# B&R Automation Studio project dbserv_0640 (part 12)

#### brtcp.c
```c
#ifdef _DEFAULT_INCLUDES
	#include <AsDefault.h>
#endif
/*************************************************************************************************
	Treiber für TCP/IP-Kopplung zwischen zenOn und brserver

	Stand:		11.04.03
	Verfasser:	L.Waibel, MEGASYSTEMS GmbH
    LastEdit:

        21.12.04/RES:	#include von bsrun.h bzw. dbserv.h durch Compilerschalter geregelt
        11.12.04/RES:	Fehler bei ClientCommands() - case BRT_ITM_READ beseitigt
        08.12.03/Wai:	Fehler bei ITEM_WRITE ohne vorheriges LOGON behoben
		06.07.04/WAI:	Diagnose wegen Abstürzen mit divide-error
						(ClientDiag = protokollieren aller Client-Anmeldungen, ClientsMax=max.Anzahl Clients,
						Verwendung der max.Anzahl Clients aus dplist, statt MAX_CLIENTS
    	13.08.03/RES:	Diagnose-PVs reduziert; ClientDiagnose() eingefuegt ( nur fuer Burklimat2000 )
 		11.08.03/RES:	Alle "i" ersetzt durch "clientNr"
        15.07.03/RES:	Diagnosen eingebaut DIAG_*
                        Fehler bei ClientRecv() und ClientCommands() beseitigt
		08.09.06/WAI:	ClientConnect() Client möglichst wieder bei gleicher Instanz anmelden
						wegen Archivierung
		18.02.15/BIE:	Erweiterung für ATOM-CPUs

**************************************************************************************************/

#define _REPLACE_CONST		//18.02.2015 Erweiterung für ATOM-CPUs
#define ETH_SOCK_NG 1		//18.02.2015 Erweiterung für ATOM-CPUs

#include	<bur/plc.h>
#include	<bur/plctypes.h>
#include	<ethsock.h>
#include	<AsIecCon.h>
#include	<sys_lib.h>
#include	<standard.h>
#include 	<fileio.h>

#include	"platform.h"

#include	"brtcp.h"

#ifdef BURKLIMAT2000
			#include 	"bsrun.h"
			#include	"bksys.h"
#else
			#include	"dbserv.h"
#endif

/*************************************************************************************************/
/* Diagnose wegen Abstürzen */
#define	ANZAHL_CLIENTDIAG	10

typedef struct {
	UDINT		ClientAdrs;
	RTCtime_typ	LoginTime;
	UINT		LoginCount;
} CLIENTDIAG_typ;

_LOCAL	INT	ClientsMax,MaxCfgClients;
_LOCAL	CLIENTDIAG_typ	ClientDiag[ANZAHL_CLIENTDIAG];
_LOCAL	UINT	instancestate;
_LOCAL	RTCtime_typ	ActTime;

/*************************************************************************************************/
/*	globale Variablen                                                                            */
/*************************************************************************************************/

/*************************************************************************************************/
/*	lokale Variablen                                                                             */
/*************************************************************************************************/
_LOCAL	ACCESS_SERVER	*myidBrServer;

_LOCAL	UINT	idstat,brstate,portstat,timeoutstat,timeout;

_LOCAL	UINT	typestate,typecount;
_LOCAL	USINT 	step, initok;
_LOCAL	UINT	port;
_LOCAL	unsigned long	arg, socket_descr, bacllog, client_len;
_LOCAL	signed long	new_sock;
_LOCAL	int		opt_val, stat_ioctl, stat_setsockopt, stat_bind, stat_listen, clients;
_LOCAL	UINT	StateRTCTime,StateSWTime;
_LOCAL	INT		len_opt_val;

_LOCAL	ETH_sockaddr_typ name_str, client_str;
_LOCAL	INT	error;

_LOCAL	UINT	ID,AK,Anlage,Geraet,Typ,Punkt,Item;
_LOCAL	UDINT	Len,CmdLen,SendLen;

_LOCAL	CLI_HEAD_TYP *pBRT_head;
_LOCAL	CLI_LOGON_REQUEST *pBRT_logon;
_LOCAL	CLI_LOGON_RESPONSE *pBRT_logon_resp;
_LOCAL	CLI_LOGOFF_REQUEST *pBRT_logoff;
_LOCAL	CLI_LOGOFF_RESPONSE *pBRT_logoff_resp;
_LOCAL	CLI_READ_REQUEST *pBRT_read;
_LOCAL	CLI_READ_RESPONSE *pBRT_read_resp;
_LOCAL	CLI_WRITE_REQUEST *pBRT_write;
_LOCAL	CLI_WRITE_RESPONSE *pBRT_write_resp;
_LOCAL	CLI_ADRERROR_RESPONSE *pBRT_adrerror_resp;
_LOCAL	CLI_ERROR_RESPONSE *pBRT_error_resp;
_LOCAL	CLI_EVENT_RESPONSE *pBRT_event_resp;
_LOCAL	CLI_WATCHDOG_REQUEST *pBRT_watch;
_LOCAL	CLI_WATCHDOG_RESPONSE *pBRT_watch_resp;
_LOCAL	CLI_TIMESYNC_REQUEST *pBRT_time;
_LOCAL	CLI_TIMESYNC_RESPONSE *pBRT_time_resp;
_LOCAL	CLI_DATASTREAM *pBRT_datastream;

_LOCAL	client_typ	client[MAX_CLIENTS];
_LOCAL	USINT		TempBuffIn[RECVBUFLEN];
_LOCAL	USINT		TempBuffOut[SENDBUFLEN];
_LOCAL	USINT	DataByte;
_LOCAL	UINT	DataWord;
_LOCAL	UDINT	DataLong;
_LOCAL	RTCtime_typ DataTime;

_LOCAL	EVENT_PIPE_DATA	*pMSEventHeadData;

_LOCAL	unsigned char	DIAG_Init;
_LOCAL	unsigned long	DIAG_ClientAuftraege;
_LOCAL	unsigned long	DIAG_EventAuftraege;
_LOCAL	unsigned long	DIAG_LogonCount;

/***********************************************************************************************
	htons
	host to network short
***********************************************************************************************/
UINT htons(UINT in)
{
#ifndef INTEL
	return swapUINT(in);
#else
	return in;
#endif
}
/***********************************************************************************************
	htonl
	host to network long
***********************************************************************************************/
UDINT htonl(UDINT in)
{
#ifndef INTEL
	return swapUDINT(in);
#else
	return in;
#endif
}
/***********************************************************************************************
	ntohs
	network to host short
***********************************************************************************************/
UINT ntohs(UINT in)
{
#ifndef INTEL
	return swapUINT(in);
#else
	return in;
#endif
}

/***********************************************************************************************
	ntohl
	network to host long
***********************************************************************************************/
UDINT ntohl(UDINT in)
{
#ifndef INTEL
	return swapUDINT(in);
#else
	return in;
#endif
}
/***********************************************************************************************
	GetData
	kopiert plattformabhägig die Daten und stellt die korrekte Byte-Order her
	Rückgabe:	Zeiger auf die korrekten Daten
***********************************************************************************************/
void GetData( USINT *pDataSrc, USINT **pDataDest, UDINT Len)
{
	switch(Len)	{
		default:
		case 1:
			DataByte = *(USINT*)pDataSrc;
			*pDataDest = &DataByte;
			break;
		case 2:
			DataWord = ntohs(*(UINT*)pDataSrc);
			*pDataDest = (USINT*)&DataWord;
			break;
		case 4:
			DataLong = ntohl(*(UDINT*)pDataSrc);
			*pDataDest = (USINT*)&DataLong;
			break;
		case sizeof(RTCtime_typ):
			memcpy((USINT*)&DataTime,pDataSrc,Len);
			DataTime.year = ntohs(DataTime.year);
			*pDataDest = (USINT*)&DataTime;
			break;
	}
}

/***********************************************************************************************
	TcpError
	kodiert die Meldeserver-Fehlernummern auf TCP-Fehlernummern um
***********************************************************************************************/
UINT TcpError(UINT inerror)
{
	UINT	outerror;

	switch (inerror)	{
		case cEC_INVALID_UNIT:
			outerror = BRT_ERR_UNKNOWN_UNIT;
			break;
		case cEC_INVALID_DEVICE:
			outerror = BRT_ERR_UNKNOWN_DEVICE;
			break;
		case cEC_INVALID_TYPE:
			outerror = BRT_ERR_UNKNOWN_TYPE;
			break;
		case cEC_INVALID_POINT:
			outerror = BRT_ERR_UNKNOWN_POINT;
			break;
		case cEC_INVALID_ITEM:
			outerror = BRT_ERR_WRONG_ITEM;
			break;
		case cEC_INVALID_LENGTH:
			outerror = BRT_ERR_WRONG_LEN;
			break;
		case cEC_ITEM_ALREADY_LINKED:
			outerror = BRT_ERR_IS_LOGGED;
			break;
		case cEC_ITEM_ALREADY_UNLINKED:
			outerror = BRT_ERR_ITEM_NO_LOGON;
			break;
		case cEC_ITEM_NOT_WRITEABLE:
			outerror = BRT_ERR_ITEM_NOT_WRITEABLE;
			break;
		case cEC_WRITE_PIPE_FULL:
			outerror = BRT_ERR_WRITE_PIPE_FULL;
			break;
		case cEC_ITEM_NO_TIMESTAMP:
			outerror = BRT_ERR_ITEM_NO_TS;
			break;
		case cEC_INVALID_VALUE:
			outerror = BRT_ERR_ITEM_NO_DATA;
			break;
		default:
			outerror = inerror;
			break;
	}
	return outerror;
}
/***********************************************************************************************
	GetAdrs
	liest die aktuelle Adresse aus dem Telegramm in Einzelvariablen
***********************************************************************************************/
void GetAdrs(CLI_ADR_TYP *pAdrs)
{
	Anlage = ntohs(pAdrs->anlage);
	Geraet = ntohs(pAdrs->geraet);
	Typ = ntohs(pAdrs->typ);
	Punkt = ntohs(pAdrs->punkt);
	Item = ntohs(pAdrs->item);
}
/***********************************************************************************************
	PutAdrs
	schreibt die aktuelle Adresse in das Telegramm aus Einzelvariablen
***********************************************************************************************/
void PutAdrs(CLI_ADR_TYP *pAdrs)
{
	pAdrs->anlage = htons(Anlage);
	pAdrs->geraet = htons(Geraet);
	pAdrs->typ = htons(Typ);
	pAdrs->punkt = htons(Punkt);
	pAdrs->item = htons(Item);
}
/***********************************************************************************************
	NextCmd
	schaltet Empfangspuffer auf nächsten Befehl und setzt ggf. Puffer zurück
***********************************************************************************************/
void NextCmd(INT clientNr, UDINT len)
{
	client[clientNr].recv_out += len;
	if(client[clientNr].recv_out == client[clientNr].recv_in)	{
		client[clientNr].recv_out = client[clientNr].recv_in = 0;		/* reset buffer */
	}
}
/***********************************************************************************************
	SpaceSendBuf
	prüft, ob die angeforderte Datenlänge noch in den Sendepuffer passt
***********************************************************************************************/
int SpaceSendBuf(INT clientNr, UDINT len)
{
	return( (sizeof(client[clientNr].send_buf) - client[clientNr].send_in) > len ? 1:0);
}

/***********************************************************************************************
	ClientConnect
	akzeptiert neue Client-Verbindungen
***********************************************************************************************/
void ClientConnect()
{
	INT	clientNr;
	BOOL new_client;
	BOOL old_entry;

	new_client = FALSE;
	client_len = sizeof(client_str);
	new_sock = accept(socket_descr, (unsigned long)&client_str, (unsigned long)&client_len);
	if (new_sock != ERR_SOCKET)	{
		/* new connection */
		for(clientNr=0;clientNr<MaxCfgClients;clientNr++)	{		/* 06.07.04: statt MAX_CLIENTS */
			/* 08.09.06: gleichen Client über IP-Adrs möglichst an gleicher Instanz anmelden wegen Archivierung */
			if(client[clientNr].socket==ERR_SOCKET && client[clientNr].client_str.sin_addr == client_str.sin_addr)	{
				/* new client */
				client[clientNr].socket = new_sock;
				client[clientNr].recv_in = 0;
				client[clientNr].recv_out = 0;
				client[clientNr].send_in = 0;
				client[clientNr].send_out = 0;
				client[clientNr].status = CLI_CONNECTED;
				client[clientNr].TON_watchdog.IN = FALSE;
				client[clientNr].stateEvRead = cEC_NO_DATA_IN_EVENTBUFFER;
				clients++;
				/* 06.07.04: save ClientsMax */
				if(clients > ClientsMax)	ClientsMax = clients;

				new_client = TRUE;
				memcpy(&client[clientNr].client_str,&client_str,sizeof(client_str));
				break;
			}
		}
		if(!new_client)	{
			/* 08.09.06: falls Client noch nie angemeldet war: nächsten freien Client nehmen */
			for(clientNr=0;clientNr<MaxCfgClients;clientNr++)	{		/* 06.07.04: statt MAX_CLIENTS */
				if(client[clientNr].socket==ERR_SOCKET)	{
					/* new client */
					client[clientNr].socket = new_sock;
					client[clientNr].recv_in = 0;
					client[clientNr].recv_out = 0;
					client[clientNr].send_in = 0;
					client[clientNr].send_out = 0;
					client[clientNr].status = CLI_CONNECTED;
					client[clientNr].TON_watchdog.IN = FALSE;
					client[clientNr].stateEvRead = cEC_NO_DATA_IN_EVENTBUFFER;
					clients++;
					/* ArchiveFiles löschen bei neuem Client */

					/* 06.07.04: save ClientsMax */
					if(clients > ClientsMax)	ClientsMax = clients;

					new_client = TRUE;
					memcpy(&client[clientNr].client_str,&client_str,sizeof(client_str));
					break;
				}
			}
		}
		/*---------------------------------------------------------------------------*/
		/* 06.07.04: diagnostics: log every connecting client */
		old_entry = 0;
		for(clientNr=0;clientNr< ANZAHL_CLIENTDIAG;clientNr++)	{
			if(ClientDiag[clientNr].ClientAdrs == client_str.sin_addr)	{
				RTC_gettime(&ActTime);
				memcpy(&ClientDiag[clientNr].LoginTime,&ActTime,sizeof(ActTime));
				ClientDiag[clientNr].LoginCount++;
				old_entry = TRUE;
				break;
			}
		}
		if(!old_entry)	{
			/* look for new entry in list */
			for(clientNr=0;clientNr< ANZAHL_CLIENTDIAG;clientNr++)	{
				if(ClientDiag[clientNr].ClientAdrs == 0 || clientNr == ANZAHL_CLIENTDIAG-1)	{	/* auf jeden in letztem Platz eintragen */
					RTC_gettime(&ActTime);
					ClientDiag[clientNr].ClientAdrs = client_str.sin_addr;
					memcpy(&ClientDiag[clientNr].LoginTime,&ActTime,sizeof(ActTime));
					ClientDiag[clientNr].LoginCount++;
					break;
				}
			}
		}
		/* 06.07.04: end diagnostics: log every connecting client */
		/*---------------------------------------------------------------------------*/

		if(!new_client)	{
			close(new_sock);		/* immediately terminate new connection */
		}
	}
}
/***********************************************************************************************
	ClientClose
	beendet Verbindung zu einem Client
***********************************************************************************************/
void ClientClose(INT clientNr, INT reason)
{
	close(client[clientNr].socket);
	client[clientNr].socket = ERR_SOCKET;
	client[clientNr].status = reason;
	client[clientNr].TON_watchdog.IN = FALSE;
/*	UnlinkEventInstance(myidBrServer,clientNr);*/
	UnlinkEventInstanceWithoutFileBuffer(myidBrServer,clientNr);		/* WAI 09.04.06 */
	if(clients)	clients--;
}
/***********************************************************************************************
	ClientWatch
	prüft auf Verbindungstimeout zu einem Client
***********************************************************************************************/
void ClientWatch(INT clientNr)
{
	TON(&client[clientNr].TON_watchdog);
	client[clientNr].TON_watchdog.IN = TRUE;
	if(client[clientNr].TON_watchdog.Q == TRUE)	{
		/* Timeout !	close connection */
		ClientClose(clientNr,CLI_WATCHDOG);
	}
}

/***********************************************************************************************
	ClientRecv
	empfängt Daten von den aktiven Clients
***********************************************************************************************/
UDINT ClientRecv(INT clientNr)
{
	DINT	bytes = 0;		/* 15.07.03/RES: bytes = 0 */
	UDINT	recv_len;

	/* read data from client */
	recv_len = sizeof(client[clientNr].recv_buf) - client[clientNr].recv_in;
	if( recv_len > 0 ) {		/* 15.07.03/RES */
		bytes = recv(client[clientNr].socket,(UDINT)&client[clientNr].recv_buf[client[clientNr].recv_in],recv_len,0);
		if(bytes==0)	{
			/* connection closed */
			ClientClose(clientNr,CLI_DISCONNECTED);
		}
		else if(bytes == ERR_SOCKET){
			/* error */
			error = EthGetError();
			if(error != ERR_ETH_WOULDBLOCK )	{
				/* all errors except: waiting for data */
				ClientClose(clientNr,CLI_ERROR);
			}
		}
		else {
			/* data received */
			client[clientNr].recv_cnt++;
			client[clientNr].TON_watchdog.IN = FALSE;
			client[clientNr].recv_in +=bytes;
		}
	}
	return bytes;
}
/***********************************************************************************************
	ClientCommands
	wertet die Kommandos eines Clients aus
***********************************************************************************************/
void ClientCommands(INT clientNr)
{
	BOOL	wait_data = FALSE;
	UDINT	shiftlen,TempLen;
	UINT	mserror = 0;
	USINT	*pData,*pTime,*pDest;
	UDINT	lenData,lenTime;

	if(client[clientNr].recv_in  < (client[clientNr].recv_out+sizeof(CLI_HEAD_TYP))) {
		wait_data = TRUE;		/* no data */
	}
	else {
		do	{

			memcpy(TempBuffIn,&client[clientNr].recv_buf[client[clientNr].recv_out],client[clientNr].recv_in - client[clientNr].recv_out);
			pBRT_head = (CLI_HEAD_TYP *)TempBuffIn;
			ID  = ntohs(pBRT_head->ID);
			AK	= ntohs(pBRT_head->AK);

			DIAG_ClientAuftraege++;

			switch(AK)	{
				/*...........................................................................................*/
				/* Item mit/ohne Zeitstempel anmelden */
				case BRT_ITM_LOGON:
				case BRT_ITM_LOGON_TS:
					if(client[clientNr].recv_in  >= (client[clientNr].recv_out+sizeof(CLI_LOGON_REQUEST)-2))	{
						pBRT_logon = (CLI_LOGON_REQUEST *)pBRT_head;
						Len = (UDINT)ntohs(pBRT_logon->LenHigh)<<16 | ntohs(pBRT_logon->LenLow) ;
						CmdLen = sizeof(CLI_LOGON_REQUEST)+ Len - 2;
						if(client[clientNr].recv_in  >= client[clientNr].recv_out + CmdLen)	{
							GetAdrs(&pBRT_logon->Adr);		/* Adresse aus Telegramm lesen */

							if(AK == BRT_ITM_LOGON)
								SendLen = CmdLen;						/* LOGON_RESPONSE max. gleich lang wie REQUEST ! */
							else
								SendLen = CmdLen +sizeof(RTCtime_typ);	/* LOGON_RESPONSE max. gleich lang wie REQUEST ! */

							if(SpaceSendBuf(clientNr, SendLen))	{	/* Platz in Sendepuffer vorhanden ?*/

								DIAG_LogonCount++;

								/* Hysterese kopieren */
								GetData((USINT*)&pBRT_logon->Data,(USINT**)&pData,Len);	/* Daten ggf. swappen */
								if((mserror = SetHystItem (myidBrServer,clientNr,Anlage,Geraet,Typ,Punkt,Item,pData,Len))==0)	{
									/* Datenpunkt anmelden */
									mserror=LinkEventItem(myidBrServer,clientNr,Anlage,Geraet,Typ,Punkt,Item,(AK == BRT_ITM_LOGON ? 0:1));
									if(mserror == 0 || mserror == cEC_ITEM_ALREADY_LINKED_FILE_BUFFER)	{	/* wegen Langzeitarchivierung */
										/* AktWert besorgen */
										mserror = GetValueItem (myidBrServer,clientNr, Anlage, Geraet, Typ, Punkt, Item, &pData, &lenData, &pTime, &lenTime);
									}
									if(mserror == 0)	{
										if( Len != lenData || (AK==BRT_ITM_LOGON_TS && lenTime==0))	{
											/* falsche Länge oder kein Zeitstempel vorhanden */
											if(Len != lenData)	mserror = BRT_ERR_WRONG_LEN;
											else				mserror = BRT_ERR_ITEM_NO_TS;

											pBRT_adrerror_resp = (CLI_ADRERROR_RESPONSE *)TempBuffOut;
											pBRT_adrerror_resp->head.ID = htons(ID);
											pBRT_adrerror_resp->head.AK = htons(BRT_ITM_LOGON_ERR);
											PutAdrs(&pBRT_adrerror_resp->Adr);
											pBRT_adrerror_resp->Error = htons(TcpError(mserror));
											SendLen = sizeof(CLI_ADRERROR_RESPONSE);
										}
										else {
											/* Sendedaten bereitstellen */
											pBRT_logon_resp = (CLI_LOGON_RESPONSE *)&TempBuffOut;
											pBRT_logon_resp->head.ID = htons(ID);
											PutAdrs(&pBRT_logon_resp->Adr);

											if(AK == BRT_ITM_LOGON)	{
												pBRT_logon_resp->head.AK = htons(BRT_ITM_LOGON_OK);
											}
											else	{
												pBRT_logon_resp->head.AK = htons(BRT_ITM_LOGON_TS_OK);
											}
											TempLen = htonl(lenData);
											memcpy(&pBRT_logon_resp->LenLow,&TempLen,sizeof(TempLen));
											/* Daten kopieren */
											GetData(pData,(USINT**)&pDest,lenData);
											memcpy(&pBRT_logon_resp->Data,pDest,lenData);
											/* ggf. Zeitstempel kopieren */
											if(AK == BRT_ITM_LOGON_TS)	{
												GetData(pTime,(USINT**)&pDest,lenTime);
												memcpy((USINT*)&pBRT_logon_resp->Data+lenData,pDest,lenTime);
											}
										}
									}
									else {	/* Fehler beim Lesen des Datenpunkts */
										/* Sendedaten bereitstellen */
										pBRT_adrerror_resp = (CLI_ADRERROR_RESPONSE *)TempBuffOut;
										pBRT_adrerror_resp->head.ID = htons(ID);
										pBRT_adrerror_resp->head.AK = htons(BRT_ITM_LOGON_ERR);
										PutAdrs(&pBRT_adrerror_resp->Adr);
										pBRT_adrerror_resp->Error = htons(TcpError(mserror));
										SendLen = sizeof(CLI_ADRERROR_RESPONSE);
									}
								}
								else {	/* logon-error */
									/* Sendedaten bereitstellen */
									pBRT_adrerror_resp = (CLI_ADRERROR_RESPONSE *)TempBuffOut;
									pBRT_adrerror_resp->head.ID = htons(ID);
									pBRT_adrerror_resp->head.AK = htons(BRT_ITM_LOGON_ERR);
									PutAdrs(&pBRT_adrerror_resp->Adr);
									pBRT_adrerror_resp->Error = htons(TcpError(mserror));

									SendLen = sizeof(CLI_ADRERROR_RESPONSE);
								}
								memcpy(&client[clientNr].send_buf[client[clientNr].send_in],TempBuffOut,SendLen);
								client[clientNr].send_in += SendLen;
								/* goto next command */
								NextCmd(clientNr, CmdLen);
							}
							else	wait_data = TRUE;	/* wait for sendbuffer free */
						}
						else wait_data = TRUE;	/* incomplete data */
					}
					else wait_data = TRUE;	/* incomplete data */
					break;
				/*...........................................................................................*/
				/* Item abmelden */
				case BRT_ITM_LOGOFF:
					CmdLen = sizeof(CLI_LOGOFF_REQUEST);
					if(client[clientNr].recv_in  >= client[clientNr].recv_out + CmdLen)	{
						pBRT_logoff = (CLI_LOGOFF_REQUEST *)pBRT_head;
						GetAdrs(&pBRT_logoff->Adr);		/* Adresse aus Telegramm lesen */

						SendLen = sizeof(CLI_ADRERROR_RESPONSE);	/* LOGOFF_RESPONSE max. gleich lang wie ADRERROR_RESPONSE ! */

						if(SpaceSendBuf(clientNr, SendLen))	{	/* Platz in Sendepuffer vorhanden ?*/
							if((error=UnlinkEventItem(myidBrServer,clientNr,Anlage,Geraet,Typ,Punkt,Item))==0)	{
								/* Sendedaten bereitstellen */
								pBRT_logoff_resp = (CLI_LOGOFF_RESPONSE *)TempBuffOut;
								pBRT_logoff_resp->head.ID = htons(ID);
								pBRT_logoff_resp->head.AK = htons(BRT_ITM_LOGOFF_OK);
								PutAdrs(&pBRT_logoff_resp->Adr);
								SendLen = CmdLen;
							}
							else {	/* logoff-error */
								/* Sendedaten bereitstellen */
								pBRT_adrerror_resp = (CLI_ADRERROR_RESPONSE *)TempBuffOut;
								pBRT_adrerror_resp->head.ID = htons(ID);
								pBRT_adrerror_resp->head.AK = htons(BRT_ITM_LOGOFF_ERR);
								PutAdrs(&pBRT_adrerror_resp->Adr);
								pBRT_adrerror_resp->Error = htons(TcpError(error));
								SendLen = sizeof(CLI_ADRERROR_RESPONSE);
							}
							memcpy(&client[clientNr].send_buf[client[clientNr].send_in],TempBuffOut,SendLen);
							client[clientNr].send_in += SendLen;
							/* goto next command */
							NextCmd(clientNr, CmdLen);
						}
						else	wait_data = TRUE;	/* wait for sendbuffer free */
					}
					else wait_data = TRUE;	/* incomplete data */
					break;
				/*...........................................................................................*/
				/* Item mit/ohne Zeitstempel lesen */
				case BRT_ITM_READ:
				case BRT_ITM_READ_TS:
					CmdLen = sizeof(CLI_READ_REQUEST);
					if(client[clientNr].recv_in  >= client[clientNr].recv_out + CmdLen)	{
						pBRT_read = (CLI_READ_REQUEST *)pBRT_head;
						GetAdrs(&pBRT_read->Adr);		/* Adresse aus Telegramm lesen */

						/* AktWert besorgen */
						mserror = GetValueItem (myidBrServer,clientNr, Anlage, Geraet, Typ, Punkt, Item, &pData, &lenData, &pTime, &lenTime);
						if(mserror == 0)	{
							if(AK==BRT_ITM_READ)
								SendLen = sizeof(CLI_READ_RESPONSE)+lenData-2;
							else
								SendLen = sizeof(CLI_READ_RESPONSE)+lenData-2+sizeof(RTCtime_typ);

							if(SpaceSendBuf(clientNr, SendLen))	{	/* Platz in Sendepuffer vorhanden ?*/
								if(AK==BRT_ITM_READ_TS && lenTime==0)	{
								/* kein Zeitstempel vorhanden */
									mserror = BRT_ERR_ITEM_NO_TS;

									pBRT_adrerror_resp = (CLI_ADRERROR_RESPONSE *)TempBuffOut;
									pBRT_adrerror_resp->head.ID = htons(ID);
									pBRT_adrerror_resp->head.AK = htons(BRT_ITM_READ_ERR);
									PutAdrs(&pBRT_adrerror_resp->Adr);
									pBRT_adrerror_resp->Error = htons(TcpError(mserror));
									SendLen = sizeof(CLI_ADRERROR_RESPONSE);
								}
								else {
									/* Sendedaten bereitstellen */
									pBRT_read_resp = (CLI_READ_RESPONSE *)&TempBuffOut;
									pBRT_read_resp->head.ID = htons(ID);
									PutAdrs(&pBRT_read_resp->Adr);

									if(AK == BRT_ITM_READ)	{
										pBRT_read_resp->head.AK = htons(BRT_ITM_READ_OK);
									}
									else	{
										pBRT_read_resp->head.AK = htons(BRT_ITM_READ_TS_OK);
										Len += sizeof(RTCtime_typ);
									}
									TempLen = htonl(lenData);	/* wegen alignment UDINT ! */
									memcpy(&pBRT_read_resp->LenLow,&TempLen,sizeof(TempLen));
									/* Daten kopieren */
									GetData(pData,(USINT**)&pDest,lenData);
									memcpy(&pBRT_read_resp->Data,pDest,lenData);
									/* ggf. Zeitstempel kopieren */
									if(AK == BRT_ITM_READ_TS) {						/* 11.12.04/RES: hier fehlende Klammern eingefuegt !! */
										GetData(pTime,(USINT**)&pDest,lenTime);
										memcpy((USINT*)&pBRT_read_resp->Data+lenData,pDest,lenTime);
									}
								}
								memcpy(&client[clientNr].send_buf[client[clientNr].send_in],TempBuffOut,SendLen);
								client[clientNr].send_in += SendLen;
								/* goto next command */
								NextCmd(clientNr, CmdLen);
							}
							else wait_data = TRUE;	/* wait for sendbuffer free */
						}
						else	{	/* Fehler beim Lesen des Datenpunkts */
							SendLen = sizeof(CLI_ADRERROR_RESPONSE);
							if(SpaceSendBuf(clientNr, SendLen))	{	/* Platz in Sendepuffer vorhanden ?*/
								pBRT_adrerror_resp = (CLI_ADRERROR_RESPONSE *)TempBuffOut;
								pBRT_adrerror_resp->head.ID = htons(ID);
								pBRT_adrerror_resp->head.AK = htons(BRT_ITM_LOGON_ERR);
								PutAdrs(&pBRT_adrerror_resp->Adr);
								pBRT_adrerror_resp->Error = htons(TcpError(mserror));

								memcpy(&client[clientNr].send_buf[client[clientNr].send_in],TempBuffOut,SendLen);
								client[clientNr].send_in += SendLen;
								/* goto next command */
								NextCmd(clientNr, CmdLen);
							}
							else wait_data = TRUE;	/* wait for sendbuffer free */
						}
					}
					else wait_data = TRUE;	/* incomplete data */
					break;
				/*...........................................................................................*/
				/* Item schreiben */
				case BRT_ITM_WRITE:
					if(client[clientNr].recv_in  >= (client[clientNr].recv_out+sizeof(CLI_WRITE_REQUEST)-2))	{
						pBRT_write = (CLI_WRITE_REQUEST *)pBRT_head;
						Len = (UDINT)ntohs(pBRT_write->LenHigh)<<16 | ntohs(pBRT_write->LenLow) ;
						CmdLen = sizeof(CLI_WRITE_REQUEST)+ Len - 2;
						if(client[clientNr].recv_in  >= client[clientNr].recv_out + CmdLen)	{
							GetAdrs(&pBRT_write->Adr);		/* Adresse aus Telegramm lesen */

							SendLen = sizeof(CLI_ADRERROR_RESPONSE);	/* WRITE_RESPONSE max. gleich lang wie ADRERROR_RESPONSE ! */

							if(SpaceSendBuf(clientNr, SendLen))	{	/* Platz in Sendepuffer vorhanden ?*/
								GetData((USINT*)&pBRT_write->Data,(USINT**)&pData,Len);	/* Daten ggf. swappen */
								mserror = SetWriteItem(myidBrServer,Anlage,Geraet,Typ,Punkt,Item,pData,Len);

								if(mserror==0)	{
									/* Sendedaten bereitstellen */
									pBRT_write_resp = (CLI_WRITE_RESPONSE *)TempBuffOut;
									pBRT_write_resp->head.ID = htons(ID);
									PutAdrs(&pBRT_write_resp->Adr);
									pBRT_write_resp->head.AK = htons(BRT_ITM_WRITE_OK);
									SendLen = sizeof(CLI_WRITE_RESPONSE);
								}
								else {	/* write-error */
									/* Sendedaten bereitstellen */
									pBRT_adrerror_resp = (CLI_ADRERROR_RESPONSE *)TempBuffOut;
									pBRT_adrerror_resp->head.ID = htons(ID);
									pBRT_adrerror_resp->head.AK = htons(BRT_ITM_WRITE_ERR);
									PutAdrs(&pBRT_adrerror_resp->Adr);
									pBRT_adrerror_resp->Error = htons(TcpError(mserror));
									SendLen = sizeof(CLI_ADRERROR_RESPONSE);
								}
								memcpy(&client[clientNr].send_buf[client[clientNr].send_in],TempBuffOut,SendLen);
								client[clientNr].send_in += SendLen;
								/* goto next command */
								NextCmd(clientNr, CmdLen);
							}
							else	wait_data = TRUE;	/* wait for sendbuffer free */
						}
						else wait_data = TRUE;	/* incomplete data */
					}
					else wait_data = TRUE;	/* incomplete data */
					break;
				/*...........................................................................................*/
				/* Datenstrom lesen */
				case BRT_DATASTREAM_READ:
					CmdLen = sizeof(CLI_READ_REQUEST);
					if(client[clientNr].recv_in  >= client[clientNr].recv_out + CmdLen)	{
						pBRT_read = (CLI_READ_REQUEST *)pBRT_head;
						GetAdrs(&pBRT_read->Adr);		/* Adresse aus Telegramm lesen */

						/* Sonderbehandlung fehlt noch . eigener Buffer, eigenes Flag .. */
						/* AktWert besorgen */
						/*mserror = get_station_type_point (idMessageServer, Geraet, Typ, Punkt, &pData, &lenData, 0, 0, &pTime, &lenTime, 0, 0);*/
						if(mserror == 0)	{
							SendLen = sizeof(CLI_READ_RESPONSE)+lenData-2;

							if(SpaceSendBuf(clientNr, SendLen))	{	/* Platz in Sendepuffer vorhanden ?*/
								/* Sendedaten bereitstellen */
								pBRT_read_resp = (CLI_READ_RESPONSE *)&TempBuffOut;
								pBRT_read_resp->head.ID = htons(ID);
								PutAdrs(&pBRT_read_resp->Adr);

								pBRT_read_resp->head.AK = htons(BRT_DATASTREAM_READ_OK);

								TempLen = htonl(lenData);	/* wegen alignment UDINT ! */
								memcpy(&pBRT_read_resp->LenLow,&TempLen,sizeof(TempLen));
								/* Daten kopieren */
								memcpy(&pBRT_read_resp->Data,pData,lenData);

								memcpy(&client[clientNr].send_buf[client[clientNr].send_in],TempBuffOut,SendLen);
								client[clientNr].send_in += SendLen;
								/* goto next command */
								NextCmd(clientNr, CmdLen);
							}
							else wait_data = TRUE;	/* wait for sendbuffer free */
						}
						else	{	/* Fehler beim Lesen des Datenpunkts */
							SendLen = sizeof(CLI_ADRERROR_RESPONSE);
							if(SpaceSendBuf(clientNr, SendLen))	{	/* Platz in Sendepuffer vorhanden ?*/
								pBRT_adrerror_resp = (CLI_ADRERROR_RESPONSE *)TempBuffOut;
								pBRT_adrerror_resp->head.ID = htons(ID);
								pBRT_adrerror_resp->head.AK = htons(BRT_DATASTREAM_READ_ERR);
								PutAdrs(&pBRT_adrerror_resp->Adr);
								pBRT_adrerror_resp->Error = htons(TcpError(mserror));
							}
							else wait_data = TRUE;	/* wait for sendbuffer free */
						}
					}
					else wait_data = TRUE;	/* incomplete data */
					break;
				/*...........................................................................................*/
				/* Watchdog */
				case BRT_CLI_WATCHDOG:
					CmdLen = sizeof(CLI_WATCHDOG_REQUEST);
					if(client[clientNr].recv_in  >= client[clientNr].recv_out + CmdLen)	{
						pBRT_watch = (CLI_WATCHDOG_REQUEST *)pBRT_head;
						SendLen = sizeof(CLI_WATCHDOG_RESPONSE);

						if(SpaceSendBuf(clientNr, SendLen))	{	/* Platz in Sendepuffer vorhanden ?*/
							/* Sendedaten bereitstellen */
							pBRT_watch_resp = (CLI_WATCHDOG_RESPONSE *)TempBuffOut;
							pBRT_watch_resp->head.ID = htons(ID);
							pBRT_watch_resp->head.AK = htons(BRT_CLI_WATCHDOG_OK);
							memcpy(&client[clientNr].send_buf[client[clientNr].send_in],TempBuffOut,SendLen);
							client[clientNr].send_in += SendLen;
							/* goto next command */
							NextCmd(clientNr, CmdLen);
						}
						else	wait_data = TRUE;	/* wait for sendbuffer free */
					}
					else wait_data = TRUE;	/* incomplete data */
					break;
				/*...........................................................................................*/
				/* Zeitsynchronisation */
				case BRT_TIMESYNC:
					CmdLen = sizeof(CLI_TIMESYNC_REQUEST);
					if(client[clientNr].recv_in  >= client[clientNr].recv_out + CmdLen)	{
						pBRT_time = (CLI_TIMESYNC_REQUEST *)pBRT_head;
						SendLen = sizeof(CLI_ERROR_RESPONSE);		/* max.Antwortlänge */

						if(SpaceSendBuf(clientNr, SendLen))	{	/* Platz in Sendepuffer vorhanden ?*/
							/* Echtzeituhr stellen */
							pBRT_time->Time.year = ntohs(pBRT_time->Time.year );
							pBRT_time->Time.reserve = 0;
/*							pBRT_time->Time.millisec = 0;
							pBRT_time->Time.microsec = 0;*/
							StateRTCTime = RTC_settime(&pBRT_time->Time);
	#ifndef INTEL
							StateSWTime = SW_settime(&pBRT_time->Time);
	#else
							StateSWTime = 0;
	#endif

							if(StateRTCTime==0 && StateSWTime==0)	{
								/* Sendedaten bereitstellen */
								pBRT_time_resp = (CLI_TIMESYNC_RESPONSE *)TempBuffOut;
								pBRT_time_resp->head.ID = htons(ID);
								pBRT_time_resp->head.AK = htons(BRT_TIMESYNC_OK);
								SendLen = sizeof(CLI_TIMESYNC_RESPONSE );
							}
							else {	/* Fehler bei Uhrzeit stellen */
								pBRT_error_resp = (CLI_ERROR_RESPONSE *)TempBuffOut;
								pBRT_error_resp->head.ID = htons(ID);
								pBRT_error_resp->head.AK = htons(BRT_TIMESYNC_ERR);
								if(StateRTCTime)	pBRT_error_resp->Error = htons(BRT_ERR_RTC_SET);
								else				pBRT_error_resp->Error = htons(BRT_ERR_SWC_SET);
							}
							memcpy(&client[clientNr].send_buf[client[clientNr].send_in],TempBuffOut,SendLen);
							client[clientNr].send_in += SendLen;
							/* goto next command */
							NextCmd(clientNr, CmdLen);
						}
						else	wait_data = TRUE;	/* wait for sendbuffer free */
					}
					else wait_data = TRUE;	/* incomplete data */
					break;
				/*...........................................................................................*/
				/* unbekannte Auftragskennung */
				default:
					SendLen = sizeof(CLI_ERROR_RESPONSE);

					if(SpaceSendBuf(clientNr, SendLen))	{	/* Platz in Sendepuffer vorhanden ?*/
						/* Sendedaten bereitstellen */
						pBRT_error_resp = (CLI_ERROR_RESPONSE *)TempBuffOut;
						pBRT_error_resp->head.ID = htons(ID);
						pBRT_error_resp->head.AK = htons(BRT_CLI_ERROR);
						error = BRT_ERR_INVALIDAK;
						pBRT_error_resp->Error = htons(error);
						SendLen = sizeof(CLI_ERROR_RESPONSE);
						memcpy(&client[clientNr].send_buf[client[clientNr].send_in],TempBuffOut,SendLen);
						client[clientNr].send_in += SendLen;

						/* discard receivebuffer */
						client[clientNr].recv_in  = client[clientNr].recv_out =0;
					}
					else	wait_data = TRUE;	/* wait for sendbuffer free */
					break;
			}
		} while((client[clientNr].recv_in  > (client[clientNr].recv_out+sizeof(CLI_HEAD_TYP))) && wait_data == FALSE);
	}
	/* "verbrauchte" Daten aus Empfangspuffer entfernen d.h.: Rest an den Pufferanfang verschieben */
	if(wait_data && (client[clientNr].recv_out !=0))	{
		if(client[clientNr].recv_out > RECVBUFLEN / 4)	{
			/* nur schieben, wenn mehr als 1/4 Puffer zu schieben ist */
			shiftlen = client[clientNr].recv_in - client[clientNr].recv_out;
			memcpy(&client[clientNr].recv_buf[0],&client[clientNr].recv_buf[client[clientNr].recv_out],shiftlen);
			client[clientNr].recv_in -= client[clientNr].recv_out;
			client[clientNr].recv_out = 0;
		}
	}
}
/***********************************************************************************************
	ClientEvents
	prüft die EventPipes auf Daten
***********************************************************************************************/
void ClientEvents(INT clientNr)
{
	BOOL	wait_data = FALSE;
	INT		typ;
	UDINT	TempLen;
	EVENT_PIPE_DATA	*pEvent;
	USINT	*pData,*pTime;

	/* Events über alle Typen abfragen */
	for(typ=0;typ<typecount;typ++)	{
		do	{
			if(client[clientNr].stateEvRead !=0)		/* letztes Event abgearbeitet */
				client[clientNr].stateEvRead = GetEventItem(myidBrServer,clientNr,(client[clientNr].startType+typ)%typecount,
										client[clientNr].EventBuffer,sizeof(client[clientNr].EventBuffer),
										&client[clientNr].lenEventMessage,&client[clientNr].lengthTimeStamp);
			if(client[clientNr].stateEvRead ==0)	{
				/* Diag: Events zählen */
				client[clientNr].EventCnt++;
				/* Event vorhanden */
				pMSEventHeadData = (EVENT_PIPE_DATA*) client[clientNr].EventBuffer;
				Anlage = pMSEventHeadData->unit;
				Geraet = pMSEventHeadData->device;
				Typ = pMSEventHeadData->type;
				Punkt = pMSEventHeadData->point;
				Item = pMSEventHeadData->item;
				Len = client[clientNr].lenEventMessage;

				if( pMSEventHeadData->pData != NULL)	{
					client[clientNr].stateEvRead = cEC_NO_DATA_IN_EVENTBUFFER;
					/* Daten von Stream */
					client[clientNr].stateStream = STREAM_INIT;
					/* Abbruch wegen Start Datastream */
					wait_data = TRUE;
					break;
				}
				else {
					/* Daten aus Prozessabbild */
					SendLen = sizeof(CLI_EVENT_RESPONSE) - 2 + client[clientNr].lenEventMessage + client[clientNr].lengthTimeStamp;

					if(SpaceSendBuf(clientNr, SendLen))	{	/* Platz in Sendepuffer vorhanden ?*/
						client[clientNr].stateEvRead = cEC_NO_DATA_IN_EVENTBUFFER;
						/* Sendedaten bereitstellen */
						pBRT_event_resp = (CLI_EVENT_RESPONSE *)TempBuffOut;
						pBRT_event_resp->head.ID = htons(client[clientNr].EventID++);
						PutAdrs(&pBRT_event_resp->Adr);
						if(!client[clientNr].lengthTimeStamp)
							pBRT_event_resp->head.AK = htons(BRT_ITM_EVENT);
						else
							pBRT_event_resp->head.AK = htons(BRT_ITM_EVENT_TS);

						TempLen = htonl(Len);
						memcpy(&pBRT_event_resp->LenLow,&TempLen,sizeof(TempLen));

						/* Daten und ggf. Zeitstempel kopieren */
						pEvent = (EVENT_PIPE_DATA*)&client[clientNr].EventBuffer;
						GetData((USINT *)&client[clientNr].EventBuffer+sizeof(EVENT_PIPE_DATA),(USINT**)&pData,
								client[clientNr].lenEventMessage);
						memcpy(&pBRT_event_resp->Data, pData, client[clientNr].lenEventMessage);

						if(client[clientNr].lengthTimeStamp)	{
							GetData((USINT *)&client[clientNr].EventBuffer+sizeof(EVENT_PIPE_DATA)+client[clientNr].lenEventMessage,(USINT**)&pTime,
									client[clientNr].lengthTimeStamp);
							memcpy((USINT*)&pBRT_event_resp->Data + client[clientNr].lenEventMessage, pTime, client[clientNr].lengthTimeStamp);
						}
						/* Daten an Sendepuffer anhängen */

						DIAG_EventAuftraege++;

						memcpy(&client[clientNr].send_buf[client[clientNr].send_in],TempBuffOut,SendLen);
						client[clientNr].send_in += SendLen;
					}
					else {
						/* Abbruch wegen Überschreitung der maximalen Telegrammlänge */
						wait_data = TRUE;
					}
					break;
				}
			} /* if(client[clientNr].stateEvRead ==0) */
			else	break;
		} while (wait_data == FALSE);
		if(wait_data == TRUE)	break;
	} /*for(ev=0;ev<typecount;ev++) */

	/* Event-Abfrage um einen Typ weiterschalten */
	client[clientNr].startType  = (client[clientNr].startType+typ+1)%typecount;

}
/***********************************************************************************************
	ClientStream
	sendet Streamdaten blockweise an einen Client
***********************************************************************************************/
void ClientStream(INT clientNr)
{
	UDINT	TempLen,SendRest;

	if(client[clientNr].send_in != 0)	return;		/* wait until buffer is sent */

	switch(client[clientNr].stateStream)	{
		case STREAM_INIT:
			pMSEventHeadData = (EVENT_PIPE_DATA*) client[clientNr].EventBuffer;
			Anlage = pMSEventHeadData->unit;
			Geraet = pMSEventHeadData->device;
			Typ = pMSEventHeadData->type;
			Punkt = pMSEventHeadData->point;
			Item = pMSEventHeadData->item;
			Len = client[clientNr].lenEventMessage;

			pBRT_datastream = (CLI_DATASTREAM *)TempBuffOut;
			pBRT_datastream->head.ID = htons(client[clientNr].EventID++);
			pBRT_datastream->head.AK = htons(BRT_DATASTREAM);
			PutAdrs(&pBRT_datastream->Adr);
			TempLen = htonl(Len);
			memcpy(&pBRT_datastream->LenLow,&TempLen,sizeof(TempLen));
			/* Header in Sendebuffer eintragen */
			SendLen = sizeof(CLI_DATASTREAM);
			memcpy(&client[clientNr].send_buf[client[clientNr].send_in],TempBuffOut,SendLen);
			client[clientNr].send_in += SendLen;
			client[clientNr].stateStream = STREAM_BUSY;
			client[clientNr].pStreamData = pMSEventHeadData->pData;

		case STREAM_BUSY:
			/* Daten in Sendebuffer eintragen, bis alles gesendet ist */
			SendRest = pMSEventHeadData->pData + client[clientNr].lenEventMessage - client[clientNr].pStreamData;
			if( SendRest > (sizeof(client[clientNr].send_buf) - client[clientNr].send_in))	{
				SendLen = sizeof(client[clientNr].send_buf) - client[clientNr].send_in;
			}
			else	{
				SendLen = SendRest;
				client[clientNr].stateStream = STREAM_READY;
			}
			memcpy(&client[clientNr].send_buf[client[clientNr].send_in],client[clientNr].pStreamData,SendLen);
			client[clientNr].send_in += SendLen;
			client[clientNr].pStreamData +=SendLen;
			break;
		case STREAM_READY:
			/* Stream freigeben */
			pMSEventHeadData = (EVENT_PIPE_DATA*) client[clientNr].EventBuffer;
			Anlage = pMSEventHeadData->unit;
			Geraet = pMSEventHeadData->device;
			Typ = pMSEventHeadData->type;
			Punkt = pMSEventHeadData->point;
			Item = pMSEventHeadData->item;
/*			client[clientNr].stateRelease = ReleaseEventItemStream(myidBrServer,clientNr,Anlage,Geraet,Typ,Punkt,Item);*/

			client[clientNr].stateStream = STREAM_IDLE;
			break;
		default:
			client[clientNr].stateStream = STREAM_IDLE;
			break;
	}
}
/***********************************************************************************************
	ClientSend
	sendet Daten an einen Client
***********************************************************************************************/
void ClientSend(INT clientNr)
{
	DINT	send_len,send_ist;

	if(client[clientNr].send_in > client[clientNr].send_out)	{
		send_len = client[clientNr].send_in - client[clientNr].send_out;
		send_ist = send(client[clientNr].socket,(UDINT)&client[clientNr].send_buf[client[clientNr].send_out],send_len,0);
		if(send_ist == ERR_SOCKET)	{
			/* error */
			error = EthGetError();
			if(error != ERR_ETH_WOULDBLOCK )	{
				/* all errors except: waiting for sendbuffer free */
				ClientClose(clientNr,CLI_SENDERROR);
			}
		}
		else if (send_ist >= 0) {
			client[clientNr].send_out += send_ist;
			if(client[clientNr].send_out >= client[clientNr].send_in)	{
				client[clientNr].send_out = client[clientNr].send_in = 0;		/* total buffer was sent */
			}
		}
	}
}

/***********************************************************************************************/
_INIT void init(void)
{
	clients = 0;
	step = 0;
	initok = 0;
	DIAG_Init = 1;
}

/***********************************************************************************************/
_CYCLIC void cyclic(void)
{
	int clientNr;

	if(!initok)	{
		idstat = GetIdBrServer((void*)&myidBrServer,&brstate);
		if(!idstat)	{
			/* Portnummer holen */
			portstat = GetPortNumber(myidBrServer,&port);
			if(portstat)	{
				ERRxwarning(portstat,0,"brtcp: Portnummer ungültig");
				port = 20001;				/* Defaultwert im Fehlerfall */
			}

			/* Timeout holen */
			timeoutstat = GetTimeoutValue(myidBrServer,&timeout);
			if(timeoutstat)	{
				ERRxwarning(timeoutstat,0,"brtcp: Timeout ungültig");
				timeout = 60;				/* Defaultwert im Fehlerfall */
			}

			/* Clients initialisieren */
			for(clientNr=0;clientNr<MAX_CLIENTS;clientNr++)	{
				client[clientNr].socket = ERR_SOCKET;
				client[clientNr].status = CLI_INIT;
				client[clientNr].recv_cnt = 0;
				client[clientNr].EventCnt = 0;
				client[clientNr].TON_watchdog.PT = (UDINT)timeout * 1000;		/* [s] > [ms] */
				client[clientNr].TON_watchdog.IN = FALSE;
				TON(&client[clientNr].TON_watchdog);
				client[clientNr].stateStream = STREAM_IDLE;
			}
			initok = 1;
		}	/* idstat */
	} /* !initok */

	if(!initok)		return;

	if( DIAG_Init ) {
		DIAG_Init = 0;
		DIAG_ClientAuftraege = 0;
		DIAG_EventAuftraege = 0;
		DIAG_LogonCount = 0;
	}

	switch(step)
	{
		/*..............................................................................................*/
		/* init-states */
		case 0:
			socket_descr = socket(ETH_AF_INET, ETH_SOCK_STREAM, ETH_IPPROTO_TCP);
			if (stat_ioctl != ERR_SOCKET)	step++;
			else	{
				error = EthGetError();
				ERRxwarning(error,0,"brtcp: socket()");
				step = 255;
			}
			break;
		case 1:
			arg = 1;
			stat_ioctl = ioctl(socket_descr, ETH_FIONBIO, (unsigned long)&arg);
			if (stat_ioctl != ERR_SOCKET)	step++;
			else	{
				error = EthGetError();
				ERRxwarning(error,0,"brtcp: ioctl(ETH_FIONBIO)");
				step = 255;
			}
			break;
		case 2:
			opt_val = 1;
			len_opt_val = sizeof(opt_val);
			stat_setsockopt = setsockopt(socket_descr, ETH_SOL_SOCKET, ETH_SO_KEEPALIVE, (unsigned long)&opt_val, sizeof(opt_val));
			if (stat_setsockopt != ERR_SOCKET)	step++;
			else	{
				error = EthGetError();
				ERRxwarning(error,0,"brtcp: setsockopt(KEEPALIVE)");
				step = 255;
			}
			break;
		case 3:
			opt_val = 1;
			stat_setsockopt = setsockopt(socket_descr, ETH_SOL_SOCKET, ETH_SO_REUSEADDR, (unsigned long)&opt_val, sizeof(opt_val));
			if (stat_setsockopt != ERR_SOCKET)	step++;
			else	{
				error = EthGetError();
				ERRxwarning(error,0,"brtcp: setsockopt(REUSEADDR)");
				step = 255;
			}
			break;
		case 4:
			opt_val = sizeof(client[0].recv_buf);
			stat_setsockopt = setsockopt(socket_descr, ETH_SOL_SOCKET, ETH_SO_RCVBUF, (unsigned long)&opt_val, sizeof(opt_val));
			if (stat_setsockopt != ERR_SOCKET)	step++;
			else	{
				error = EthGetError();
				ERRxwarning(error,0,"brtcp: setsockopt(SO_RCVBUF)");
				step = 255;
			}
			break;
		case 5:
			opt_val = sizeof(client[0].send_buf);
			stat_setsockopt = setsockopt(socket_descr, ETH_SOL_SOCKET, ETH_SO_SNDBUF, (unsigned long)&opt_val, sizeof(opt_val));
			if (stat_setsockopt != ERR_SOCKET)	step++;
			else	{
				error = EthGetError();
				ERRxwarning(error,0,"brtcp: setsockopt(SO_SNDBUF)");
				step = 255;
			}
			break;
		case 6:
			name_str.sin_family = ETH_AF_INET;
#ifdef INTEL
			name_str.sin_port = swapUINT(port);
#else
			name_str.sin_port = port;
#endif
			name_str.sin_addr = MYADRS; /*(unsigned long)inet_addr((UDINT)MYADRS);*/
			memset(name_str.sin_zero,0,sizeof(name_str.sin_zero));

			stat_bind = bind(socket_descr, (unsigned long)&name_str, sizeof(name_str));
			if (stat_bind != ERR_SOCKET)	step++;
			else	{
				error = EthGetError();
				ERRxwarning(error,0,"brtcp: bind()");
				step = 255;
			}
			break;
		case 7:
			bacllog = MAX_CLIENTS;
			stat_listen = listen(socket_descr, (unsigned long)bacllog); //18.02.2015 Erweiterung für ATOM-CPUs: der Übergabeparameter bacllog muss als Variable und nicht als Zeiger übergeben werden!
			if (stat_listen != ERR_SOCKET)	step++;
			else	{
				error = EthGetError();
				ERRxwarning(error,0,"brtcp: listen()");
				step = 255;
			}
			break;
		/*..............................................................................................*/
		/* init server */
		case 8:
			if(myidBrServer!=NULL)	{
				typestate = GetTypeInfo(myidBrServer,&typecount);
				instancestate = GetEventInstanceInfo(myidBrServer,&MaxCfgClients);		/* 06.07.04 */
				if(MaxCfgClients > MAX_CLIENTS)	MaxCfgClients = MAX_CLIENTS;
				if(typestate==cEC_OK && instancestate==cEC_OK )	step++;					/* ok goto next state */
			}
			break;
		/*..............................................................................................*/
		/* working state */
		case 9:
			if(myidBrServer==NULL)	{
				/* myidBrServer invalid: goto previous state */
				step--;
				break;
			}

			ClientConnect();					/* call accept()-Funktion to connect to clients */

#ifdef BURKLIMAT2000
			ClientDiagnose();					/* Client-Diagnose ( nur Burklimat2000 ); 13.08.03/RES */
#endif

			for(clientNr=0;clientNr<MaxCfgClients;clientNr++)	{		/* 06.07.04: statt MAX_CLIENTS */
				if(client[clientNr].socket != ERR_SOCKET)	{
					ClientWatch(clientNr);		/* check for receive timeout, terminate connection */
				}
				if(client[clientNr].socket != ERR_SOCKET)	{
					if(client[clientNr].stateStream == STREAM_IDLE)	{
						ClientRecv(clientNr);		/* read frames from client */
						ClientCommands(clientNr);	/* examine client commands */
						ClientEvents(clientNr);	/* check for events */
					}
					else {
						ClientStream(clientNr);	/* send stream data */
					}
					ClientSend(clientNr);		/* send data to client (also handling of fractional sends) */
				}
			}
			break;
		/*..............................................................................................*/
		/* error state */
		case 255:
			break;
	}
}
```

#### clientdiag.c
```c
#ifdef _DEFAULT_INCLUDES
	#include <AsDefault.h>
#endif
/* clientdiag.c -------------------- */

#include <bur/plc.h>      /*some usefull macros for B&R pcc programming*/

#include <stdlib.h>

#include "bksys.h"

/*-----------------------------------------------------------------------------
// ClientDiagnose
// Berechnet diverse Diagnose-Informationen zu ClientPipes
// Last Edit:
//		13.08.03/RES:	Erstversion erstellt
//
// inputs:
// outputs:
// return:
//---------------------------------------------------------------------------*/
void ClientDiagnose( void )
{
	static	unsigned char	ClientIdx = 0;					/* Client-Index */
	static	unsigned short	Count10msOld;					/* 10ms-Taktzaehler */
	static	unsigned long	AnyPipeEntryOld[CLI_ANZ_MAX];	/* Pipe-Eintragszaehler der letzten Berechnung */
	static	unsigned long	EntryCountOld;					/* Pipe-Eintragszaehler der letzten Berechnung */

	Globals_Typ 			*pGlobals;						/* Zeiger auf Globaldatenstruktur */
	CliPipeDiagAll_Typ		*pCliPipeDiag;					/* Zeiger ClientPipe-Diagnose-Struktur */
	unsigned short			Delta10ms;						/* Vergangene Zeit in 10ms seit letzter sekuendlicher Berechnung */
	unsigned char			ClientIdxTmp;					/* Client-Index fuer temporaere Verwendung */
	unsigned char			DtIdx;							/* Datentyp-Index */
	unsigned long			EntryDiff;						/* Eintragsdifferenz */

	CliPbHead_Typ 			*pPbHead;						/* Zeiger auf Client-Pipeblock-Header */
	CliPipeHead_Typ			*pPipe;
	long					lUsed;

	/* Zeiger auf Globaldatenstruktur initialisieren */
	GetGlobalsPtr( &pGlobals );
	if( pGlobals == NULL ) {			/* Gueltige Adresse in pGlobals ? */
		return;		/* Kein gueltiger pGlobals */
	}

	/* ClientPipe-Diagnose-Monitor -------------------------------------------- */
	pCliPipeDiag = pGlobals->pCliPipeDiag;		/* Interne Datenstruktur ueber dynamische DIAG-PV (lokale Pointer PV) sichtbar machen */

	/* Initialisierung */
	if( pCliPipeDiag->Init ) {
		pCliPipeDiag->Init = 0;
		memset( pCliPipeDiag, 0, sizeof( CliPipeDiagAll_Typ ) );
	}

	/* Sekuendliche Berechnungen ---------------------------------------------- */
	Delta10ms = pGlobals->Count10ms - Count10msOld;
	if( Delta10ms >= 100 ) {
		Count10msOld = pGlobals->Count10ms;		/* Zeit abgelaufen => aktuellen 10ms Count merken */
		EntryDiff = pCliPipeDiag->EntryCount - EntryCountOld;				/* Eintragsdifferenz ermitteln */
		pCliPipeDiag->EntryCountPerSec = EntryDiff * 100 / Delta10ms;
		EntryCountOld = pCliPipeDiag->EntryCount;
		for( ClientIdxTmp = 0; ClientIdxTmp < pGlobals->pCab->ClientAnz; ClientIdxTmp++ ) {
			EntryDiff = pCliPipeDiag->Client[ClientIdxTmp].AnyPipeEntry - AnyPipeEntryOld[ClientIdxTmp];		/* Eintragsdifferenz ermitteln */
			pCliPipeDiag->Client[ClientIdxTmp].AnyPipeEntryPerSec = EntryDiff * 100 / Delta10ms;
			AnyPipeEntryOld[ClientIdxTmp] = pCliPipeDiag->Client[ClientIdxTmp].AnyPipeEntry;
		}
	}

	/* Zyklische clientweise Berechnungen ------------------------------------- */
	for( DtIdx = 0; DtIdx < DT_ANZ; DtIdx++ ) {
		lUsed = 0;
		pPbHead = pGlobals->pCab->pClientPb[ClientIdx];	/* Zeiger auf PipeBlock des angegebenen Clients ermitteln */
		if( pPbHead != 0 ) {
			pPipe = pPbHead->pDtPipe[DtIdx];	/* Zeiger auf Pipe-Header ermitteln */
			if( pPipe != 0 ) {
				/* Genutzten Platz in der Pipe berechnen */
				lUsed = pPipe->pWrite - pPipe->pRead;
				if( lUsed < 0 ) {
					lUsed += pPipe->pLast - pPipe->pFirst + 1;						/* Absolutwert */
				}
				if( pPipe->pLast > pPipe->pFirst ) {
					lUsed = ( lUsed * 100 ) / ( pPipe->pLast - pPipe->pFirst );		/* Prozentangabe */
				}
				else {
					lUsed = 0;		/* Nur sicherheitshalber !! */
				}
			}
		}
		pCliPipeDiag->Client[ClientIdx].DtPipeUse[DtIdx] = lUsed;
	}
	ClientIdx++;		/* Naechsten Client fuer naechsten Zyklus anwaehlen */
	if( ClientIdx >= pGlobals->pCab->ClientAnz ) {
		ClientIdx = 0;
	}
}
```

#### bksysbrtcp.c
```c
#ifdef _DEFAULT_INCLUDES
	#include <AsDefault.h>
#endif
/* bksysbrtcp.c --------------------------------------------------------------- */

#include <bur/plc.h>      /*some usefull macros for B&R pcc programming*/

#include <stdlib.h>			/* Standard-Library */

#include "bksys.h"

/*-----------------------------------------------------------------------------
// CliGetClientAnzMax
// Ermittelt die maximal zulaessige Clientanzahl
// Last Edit:
//		10.06.03/RES: Zeigerpruefung pCliAnzMax eingefuegt
//					  Returnwert geaendert
//		05.06.03/RES: Erstversion erstellt
//
// inputs:
//
// outputs: pCliAnzMax	Maximale Clientanzahl
//
// return:    0 kein Fehler
//			 -1 Ungueltiger pCliAnzMax-Ptr
//			-10 Kein gueltiger Globals-Ptr
//			-11 Kein gueltiger CAB-Zeiger
//---------------------------------------------------------------------------*/
short CliGetClientAnzMax( unsigned char *pCliAnzMax )
{
	Globals_Typ 	*pGlobals;		/* Zeiger auf Globaldatenstruktur */
	CabHeader_Typ	*pCab;			/* Zeiger auf CAB */

	/* Zeiger auf Struktur mit Zeigern auf Globaldaten initialisieren */
	GetGlobalsPtr( &pGlobals );

	if( pGlobals != NULL ) {	/* Gueltiger Zeiger in pGlobals ? */
		if( pCliAnzMax != NULL ) {	/* Gueltiger Zeiger in pCliAnzMax ? */
			pCab = pGlobals->pCab;
			if( pCab != NULL ) {	/* Gueltiger Zeiger in pCab ? */
				*pCliAnzMax = pCab->ClientAnz;
			}
			else {
				return( -11 );		/* Kein gueltiger CAB-Zeiger */
			}
		}
		else {
			return( -1 );		/* Kein gueltiger pCliAnzMax-Ptr */
		}
	}
	else {
		return ( -10 );		/* Kein gueltiger Globals-Ptr */
	}
	return( 0 );
}

/*-----------------------------------------------------------------------------
// CliGetDtAnz
// Ermittelt die Anzahl Datentypen
// Last Edit:
//		10.06.03/RES: Zeigerpruefung pCliAnzMax eingefuegt
//					  Returnwert geaendert
//		05.06.03/RES: Erstversion erstellt
//
// inputs:
//
// outputs: pDtAnz	Anzahl Datentypen
//
// return:    0 kein Fehler
//			 -1 Ungueltiger pDtAnz-Ptr
//---------------------------------------------------------------------------*/
short CliGetDtAnz( unsigned char *pDtAnz )
{
	if( pDtAnz != NULL ) {	/* Gueltiger Zeiger in pDtAnz ? */
		*pDtAnz = DT_ANZ;
	}
	else {
		return( -1 );		/* Kein gueltiger pDtAnz-Ptr */
	}
	return( 0 );
}

/*-----------------------------------------------------------------------------
// CliItemLink
// Setzt zum angegebenen Item das Linkflag fuer den angegebenen Client auf den
// angegebenen Status.
// Gleichzeitig wird das Logon-Flag des Clients im CAB-Header gesetzt und
// der Wert von LastVal im CAB mit dem aktuellen Itemwert initialisiert.
//
// LastEdit:
//		24.07.03/RES	Bei Link=1 nun Aktualisierung von LastVal durch AktVal (aus Alias-PV) eingefuegt
//		10.06.03/RES	Bei Link=1 nun Force-Flag=Event setzen
//		07.06.03/RES	Bei Link=1 Force-Flag=Aktualisieren (ohne Event) eingefuegt
//		02.05.03/RES	Erstversion erstellt
//
// inputs:	Client		Client-Index
//			DtIdx		Datentyp-Index
//			DpIdx		Datenpunkt-Index
//			ItemIdx		Item-Index
//			Link		Neuer Link-Status
// outputs:
// return:	  1 Item erfolgreich gelinkt
//			  0 Item hat bereits den gewuenschten Link-Status
//			 -1 Item hat keinen CAB-Eintrag
//			 -2 Unzulaessiger Client
//			 -3 Ungueltiger Datentyp
//			 -4 Unbekannter Datenpunkt
//			 -5 Unbekanntes Item
//			-10 Bk2000-Systemfehler => Globaldatenstruktur nicht gefunden
//			-11 Bk2000-Systemfehler => CAB-Header nicht gefunden
//			-12 Bk2000-Systemfehler => Dt-Props nicht gefunden
//			-13 Bk2000-Systemfehler => Dt-Desc nicht gefunden
//---------------------------------------------------------------------------*/
short CliItemLink( unsigned char Client, unsigned char DtIdx, unsigned short DpIdx, unsigned char ItemIdx, unsigned char Link )
{
	unsigned short		sRet = 0;
	Globals_Typ			*pGlobals = NULL;
	DtProps_Typ 		*pDtProps;
	DtDesc_Typ 			*pDtDesc;
	CabHeader_Typ		*pCabHead = NULL;
	unsigned char		*pPab;
	CabItemEntry_Typ	*pCab;

	/* Zeiger auf Globaldatenstruktur initialisieren */
	GetGlobalsPtr( &pGlobals );
	if( pGlobals != NULL ) {	/* Gueltiger Zeiger in pGlobals ? */
		pCabHead = pGlobals->pCab;
		if( pCabHead == NULL ) {	/* Keine gueltige Adresse in pCab ? */
			return( -11 );
		}
		/* Parameter überprüfen */
		if( Client >= pCabHead->ClientAnz ) {
			return( -2 );	/* Unzulaessiger Client */
		}
		if ( DtIdx >= DT_ANZ )	{
			return( -3 );	/* Ungueltiger Datentyp */
		}
		pDtProps = pGlobals->pDtProps + DtIdx;
		if( pDtProps == NULL ) {	/* Keine gueltige Adresse in pDtProps ? */
			return( -12 );
		}
		pDtDesc = pGlobals->pDtDesc[DtIdx];
		if( pDtDesc == NULL ) {		/* Keine gueltige Adresse in pDtDesc ? */
			return( -13 );
		}
		if ( DpIdx >= pGlobals->pPab->DpAnz[DtIdx] )	{
			return( -4 );	/* Unbekannter Datenpunkt */
		}
		if ( ItemIdx > pDtProps->DtMaxItemIdx )	{
			return( -5 );	/* Unbekanntes Item */
		}

		/* Linkflag zu Item und Client setzen ------------------------------------ */
		if( pDtDesc[ItemIdx].ItemNrCab != 0 ) {		/* Hat Item CAB-Item ? */
			pPab = pGlobals->pPab->pDtBase[DtIdx] + DpIdx * pDtProps->DtPabLen;	/* Zeiger auf DP in PAB */
			pCab = *( CabItemEntry_Typ **)( pPab + pDtProps->CabPtrOff );		/* Zeiger auf Item in CAB */
			pCab += ( pDtDesc[ItemIdx].ItemNrCab - 1 ) + ( Client * pDtProps->CabItemAnz );
			if( pCab->Link == Link ) {
				return( 0 );			/* Item hat bereits den gewuenschten Link-Status */
			}
			else {
				if( Link ) {					/* Aktionen bei Link */
					if( CliAktValToCabVal( pDtProps, pDtDesc, pPab, pCab, ItemIdx ) < 0 ) {		/* Aktuellen Wert aus Alias-PV als LastVal ins CAB schreiben */
						return( -4 );					/* Keine Alias-PV, d.h. Leiche im PAB => Fehler "Unbekannter Datenpunkt" */
					}
					pCab->Link = 1;						/* Link-Status setzen (nur, wenn aktueller Wert kopiert werden konnte) */
					pCabHead->CliLogon[Client] = 1;		/* Anmeldeflag des Clients bei Link setzen */
				}
				else {							/* Aktionen bei Unlink */
					pCab->Link = 0;						/* Link-Status loeschen */
					pCab->Force = 0;					/* Forceflag bei unlink loeschen */
				}
				sRet = 1;
			}
		}
		else {
			sRet = -1;	/* Item hat keinen CAB-Eintrag */
		}
	}
	else {
		sRet = -10;		/* Kein gueltiger Globals-Ptr */
	}
	return( sRet );
}

/*-----------------------------------------------------------------------------
// CliItemLinkAll
// Setzt fuer den angegebenen Client alle Items auf den angegebenen Status
// Gleichzeitig wird das Logon-Flag des Clients im CAB-Header gesetzt
// LastEdit:
//		25.07.03/RES	Bei Link=1 nun Aktualisierung von LastVal durch AktVal (aus Alias-PV) eingefuegt
//		10.06.03/RES	Bei Link=1 nun Force-Flag=Event setzen
//		07.06.03/RES	Bei Link=1 Force-Flag=Aktualisieren (ohne Event) eingefuegt
//		06.06.03/RES	Erstversion erstellt
//
// inputs:	Client		Client-Index
//			Link		Neuer Link-Status
// outputs:
// return:	  1 Alle Items des Clients erfolgreich gelinkt / -unlinked
//			 -1 Unzulaessiger Client
//			-10 Bk2000-Systemfehler => Globaldatenstruktur nicht gefunden
//			-11 Bk2000-Systemfehler => CAB-Header nicht gefunden
//---------------------------------------------------------------------------*/
short CliItemLinkAll( unsigned char Client, unsigned char Link )
{
	unsigned short		sRet = 0;
	Globals_Typ			*pGlobals = NULL;
	DtProps_Typ 		*pDtProps;
	DtDesc_Typ 			*pDtDesc;
	char				*pCabItemConv;
	CabHeader_Typ		*pCabHead = NULL;
	CliPipeHead_Typ		*pPipe;
	unsigned char		DtIdx;					/* Schleifenzaehler Datentypen */
	unsigned short		DpIdx;					/* Schleifenzaehler Datenpunkte */
	unsigned char		CabItemIdx;				/* Schleifenzaehler CAB-Items */
	CabItemEntry_Typ	*pCabDt, *pCabCli, *pCabDp, *pCab;
	unsigned char		*pPab;

	/* Zeiger auf Globaldatenstruktur initialisieren */
	GetGlobalsPtr( &pGlobals );
	if( pGlobals != NULL ) {	/* Gueltiger Zeiger in pGlobals ? */
		pCabHead = pGlobals->pCab;
		if( pCabHead == NULL ) {	/* Keine gueltige Adresse in pCab ? */
			return( -11 );
		}
		/* Parameter überprüfen */
		if( Client >= pCabHead->ClientAnz ) {
			return( -1 );	/* Unzulaessiger Client */
		}

		/* Bei Unlink: Zuerst Anmeldeflag des Clients loeschen */
		if( Link == 0 ) {
			pCabHead->CliLogon[Client] = 0;
		}

		/* Linkflag aller Items des Clients setzen ------------------------------------ */
		for( DtIdx = 0; DtIdx < DT_ANZ; DtIdx++ ) {		/* Schleife ueber alle Datentypen */
			pDtProps = pGlobals->pDtProps + DtIdx;
			if( pDtProps == NULL ) {		/* Keine gueltige Adresse in pDtProps ? */
				continue;
			}
			pDtDesc = pGlobals->pDtDesc[DtIdx];
			if( pDtDesc == NULL ) {			/* Keine gueltige Adresse in pDtDesc ? */
				continue;
			}
			pCabItemConv = pGlobals->pCabItemConv[DtIdx];
			if( pCabItemConv == NULL ) {	/* Keine gueltige Adresse in pCabItemConv ? */
				continue;
			}
			pCabDt = (CabItemEntry_Typ *)pCabHead->pDtBase[DtIdx];	/* Zeiger auf Datentyp im CAB */
			if( pCabDt != 0 ) {
				pCabCli = pCabDt + Client * pDtProps->CabItemAnz;	/* Zeiger auf Client im CAB */
				for( DpIdx = 0, pCabDp = pCabCli; DpIdx < pCabHead->DpAnz[DtIdx]; DpIdx++ ) {	/* Schleife ueber alle Datenpunkte dieses Datentyps */
					pPab = pGlobals->pPab->pDtBase[DtIdx] + DpIdx * pDtProps->DtPabLen;		/* Zeiger auf DP in PAB */
					for( CabItemIdx = 0, pCab = pCabDp; CabItemIdx < pDtProps->CabItemAnz; CabItemIdx++, pCab++ ) {	/* Schleife ueber alle Items dieses Datentyps */
						if( Link ) {				/* Aktionen bei Link */
							if( CliAktValToCabVal( pDtProps, pDtDesc, pPab, pCab, pCabItemConv[CabItemIdx] ) == 0 ) {	/* Aktuellen Wert aus Alias-PV als LastVal ins CAB schreiben */
								pCab->Link = 1;				/* Link-Status setzen (nur, wenn aktueller Wert kopiert werden konnte) */
							}
						}
						else {						/* Aktionen bei Unlink */
							pCab->Link = 0;					/* Link-Status loeschen */
							pCab->Force = 0;				/* Forceflag bei unlink loeschen */
						}
					}
					pCabDp += pCabHead->ClientAnz * pDtProps->CabItemAnz;
				}
			}
		}

		if( Link ) {	/* Bei Link: Zuletzt Anmeldeflag des Clients setzen */
			pCabHead->CliLogon[Client] = 1;
		}
		else {	/* Bei Unlink: Zuletzt alle Pipes des Clients leeren */
			for( DtIdx = 0; DtIdx < DT_ANZ; DtIdx++ ) {		/* Schleife ueber alle Datentypen */
				if( CliGetPipePtr( Client, DtIdx, &pPipe ) == 0 ) {
					pPipe->pRead = pPipe->pFirst;	/* Pipe leeren */
					pPipe->pWrite = pPipe->pFirst;	/* Pipe leeren */
				}
			}
		}
		sRet = 1;	/* Alles erledigt */
	}
	else {
		sRet = -10;		/* Kein gueltiger Globals-Ptr */
	}
	return( sRet );
}

/*-----------------------------------------------------------------------------
// CliSetItemHyst()
// Setzt zum angegebenen Item die Hysterese fuer den angegebenen Client
// LastEdit:
//		07.06.03/RES	Hysteresezeiger-Pruefung eingefuegt
//		02.05.03/RES	Erstversion erstellt
//
// inputs:	Client		Client-Index
//			DtIdx		Datentyp-Index
//			DpIdx		Datenpunkt-Index
//			ItemIdx		Item-Index
//			Len			Datenlaenge des Hysteresewertes
//			pHyst		Zeiger auf Hysteresewert
// outputs:
// return:	 1 = Item-Hyst erfolgreich eingetragen
//			-1 = Item hat keinen CAB-Eintrag
//			-2 = Unzulaessiger Client
//			-3 = Ungueltiger Datentyp
//			-4 = Unbekannter Datenpunkt
//			-5 = Unbekanntes Item
//			-6 = Falsche Datenlaenge
//			-7 = Ungueltiger pHyst
//			-10 = Bk2000-Systemfehler => Globaldatenstruktur nicht gefunden
//			-11 = Bk2000-Systemfehler => CAB-Header nicht gefunden
//			-12 = Bk2000-Systemfehler => Dt-Props nicht gefunden
//			-13 = Bk2000-Systemfehler => Dt-Desc nicht gefunden
//---------------------------------------------------------------------------*/
short CliSetItemHyst( unsigned char Client, unsigned char DtIdx, unsigned short DpIdx, unsigned char ItemIdx, unsigned char Len, unsigned char *pHyst )
{
	unsigned short		sRet = 0;
	Globals_Typ			*pGlobals = NULL;
	DtProps_Typ 		*pDtProps;
	DtDesc_Typ 			*pDtDesc;
	CabHeader_Typ		*pCabHead = NULL;
	unsigned char		*pPab;
	CabItemEntry_Typ	*pCab;

	GetGlobalsPtr( &pGlobals );								/* Zeiger auf Globaldatenstruktur initialisieren */
	if( pGlobals != NULL ) {
		pCabHead = pGlobals->pCab;
		if( pCabHead == NULL ) {							/* Keine gueltige Adresse in pCab ? */
			return( -11 );
		}
		if( Client >= pCabHead->ClientAnz ) {
			return( -2 );									/* Unzulaessiger Client */
		}
		if ( DtIdx >= DT_ANZ )	{
			return( -3 );									/* Ungueltiger Datentyp */
		}
		pDtProps = pGlobals->pDtProps + DtIdx;
		if( pDtProps == NULL ) {							/* Keine gueltige Adresse in pDtProps ? */
			return( -12 );
		}
		pDtDesc = pGlobals->pDtDesc[DtIdx];
		if( pDtDesc == NULL ) {								/* Keine gueltige Adresse in pDtDesc ? */
			return( -13 );
		}
		if ( DpIdx >= pGlobals->pPab->DpAnz[DtIdx] )	{
			return( -4 );									/* Unbekannter Datenpunkt */
		}
		if ( ItemIdx > pDtProps->DtMaxItemIdx )	{
			return( -5 );									/* Unbekanntes Item */
		}
		if ( Len != abs( pDtDesc[ItemIdx].ItemLen ) )	{
			return( -6 );									/* Falsche Datenlaenge */
		}
		if( pHyst == NULL ) {
			return( -7 );									/* Ungueltiger Zeiger auf Hysteresewert */
		}

		/* Hysteresewert zu Item und Client eintragen ------------------------------- */
		if( pDtDesc[ItemIdx].ItemNrCab != 0 ) {		/* Hat Item CAB-Item ? */
			pPab = pGlobals->pPab->pDtBase[DtIdx] + DpIdx * pDtProps->DtPabLen;	/* Zeiger auf DP in PAB */
			pCab = *( CabItemEntry_Typ ** )( pPab + pDtProps->CabPtrOff );		/* Zeiger auf Item in CAB */
			pCab += ( pDtDesc[ItemIdx].ItemNrCab - 1 ) + ( Client * pDtProps->CabItemAnz );
			switch( Len ) {
				case 1:
					pCab->Hyst = ( unsigned long )*pHyst;
					break;
				case 2:
					pCab->Hyst = ( unsigned long )*( unsigned short * )pHyst;
					break;
				case 4:
					pCab->Hyst = *( unsigned long * )pHyst;
					break;
				default:
					return( -6 );							/* Falsche Datenlaenge */
			}
			sRet = 1;
		}
		else {
			sRet = -1;										/* Item hat keinen CAB-Eintrag */
		}
	}
	else {
		sRet = -10;		/* Kein gueltiger Globals-Ptr */
	}

	return( sRet );
}

/*-----------------------------------------------------------------------------
// CliForceWriteEvent()
// Erzwingt zum angegebenen Item einen Event mit aktuellem Wert fuer alle gelinkten Clients
// LastEdit:
//		04.08.03/RES	Umbenannt nach CliForceWriteEvent() und Client aus Argumentliste entfernt
//		27.07.03/RES	Erstversion erstellt
//
// inputs:	DtIdx		Datentyp-Index
//			DpIdx		Datenpunkt-Index
//			ItemIdx		Item-Index
// outputs:
// return:	 1 = Event erfolgreich angefordert
//			-1 = Item hat keinen CAB-Eintrag
//			-3 = Ungueltiger Datentyp
//			-4 = Unbekannter Datenpunkt
//			-5 = Unbekanntes Item
//			-10 = Bk2000-Systemfehler => Globaldatenstruktur nicht gefunden
//			-11 = Bk2000-Systemfehler => CAB-Header nicht gefunden
//			-12 = Bk2000-Systemfehler => Dt-Props nicht gefunden
//			-13 = Bk2000-Systemfehler => Dt-Desc nicht gefunden
//---------------------------------------------------------------------------*/
short CliForceWriteEvent( unsigned char DtIdx, unsigned short DpIdx, unsigned char ItemIdx )
{
	unsigned short		sRet = 0;
	Globals_Typ			*pGlobals = NULL;
	DtProps_Typ 		*pDtProps;
	DtDesc_Typ 			*pDtDesc;
	CabHeader_Typ		*pCabHead = NULL;
	unsigned char		*pPab;
	CabItemEntry_Typ	*pCab;
	unsigned char		Client;

	GetGlobalsPtr( &pGlobals );								/* Zeiger auf Globaldatenstruktur initialisieren */
	if( pGlobals != NULL ) {
		pCabHead = pGlobals->pCab;
		if( pCabHead == NULL ) {							/* Keine gueltige Adresse in pCab ? */
			return( -11 );
		}
		if ( DtIdx >= DT_ANZ )	{
			return( -3 );									/* Ungueltiger Datentyp */
		}
		pDtProps = pGlobals->pDtProps + DtIdx;
		if( pDtProps == NULL ) {							/* Keine gueltige Adresse in pDtProps ? */
			return( -12 );
		}
		pDtDesc = pGlobals->pDtDesc[DtIdx];
		if( pDtDesc == NULL ) {								/* Keine gueltige Adresse in pDtDesc ? */
			return( -13 );
		}
		if ( DpIdx >= pGlobals->pPab->DpAnz[DtIdx] ) {
			return( -4 );									/* Unbekannter Datenpunkt */
		}
		if ( ItemIdx > pDtProps->DtMaxItemIdx )	{
			return( -5 );									/* Unbekanntes Item */
		}

		/* Hysteresewert zu Item fuer alle gelinkten Clients eintragen ------------------------------- */
		if( pDtDesc[ItemIdx].ItemNrCab != 0 ) {		/* Hat Item CAB-Item ? */
			pPab = pGlobals->pPab->pDtBase[DtIdx] + DpIdx * pDtProps->DtPabLen;	/* Zeiger auf DP in PAB */
			pCab = *( CabItemEntry_Typ ** )( pPab + pDtProps->CabPtrOff );		/* Zeiger auf Item in CAB */
			pCab += pDtDesc[ItemIdx].ItemNrCab - 1;
			for( Client = 0; Client < pCabHead->ClientAnz; Client++ ) {
				if( pCab->Link ) {
					pCab->Force = 3;	/* Event mit AKTUELLEM Wert anfordern */
				}
				pCab += pDtProps->CabItemAnz;	/* Zeiger auf Abblid fuer naechsten Client */
			}
			sRet = 1;
		}
		else {
			sRet = -1;										/* Item hat keinen CAB-Eintrag */
		}
	}
	else {
		sRet = -10;		/* Kein gueltiger Globals-Ptr */
	}

	return( sRet );
}

/*-----------------------------------------------------------------------------
// CliEvRead
// Event-Message aus Client-Event-Pipe lesen
// Last Edit:
//		08.08.03/RES: Pipe-Eintraege auf gleiche Laenge abgestimmt => schnelleres Schreiben und v.a. Lesen einer Meldung
//					  ( dabei Argumentliste geaendert )
//		07.06.03/RES: Meldungs- und Längenzeiger - Pruefung eingefuegt
//		05.06.03/RES: Erstversion aus EvRead() erzeugt
//
// inputs:	Client		Client
//			DtIdx		Datentyp-Index
//
// outputs:	pDpIdx		Datenpunkt-Index
//			pItemIdx	Item-Index
//			pItemLen	Item-Laenge
//			pValue		Item-Wert
//
// return:	  1 Meldung aus Pipe gelesen
// 			  0 keine Meldung in Pipe
//			 -1 Unzulaessiger Client
//			 -2 Unzulaessiger DtIdx
//			 -3 Unzulaessige Item-Laenge
//			<-9 Systemfehler --> siehe CliEvGetPipePtr()
//---------------------------------------------------------------------------*/
short CliEvRead( unsigned char Client, unsigned char DtIdx, unsigned short *pDpIdx, unsigned char *pItemIdx, unsigned char *pItemLen, unsigned long *pValue )
{
	short 				sRet = 0;
	CliPipeHead_Typ		*pPipe;

	if( ( sRet = CliGetPipePtr( Client, DtIdx, &pPipe ) ) == 0 ) {
		/* Daten aus Pipe in Message-Puffer kopieren */
		if( pPipe->pRead != pPipe->pWrite ) {	/* Meldung in Pipe ? */
			sRet = 1;
			*pDpIdx = pPipe->pRead->ItemAdr.DpIdx;
			*pItemIdx = pPipe->pRead->ItemAdr.ItemIdx;
			*pItemLen = pPipe->pRead->ItemAdr.ItemLen;
			switch( *pItemLen ) {
				case 1:
					*( unsigned char *)pValue = ( unsigned char )pPipe->pRead->ItemVal;
					break;
				case 2:
					*( unsigned short *)pValue = ( unsigned short )pPipe->pRead->ItemVal;
					break;
				case 4:
					*pValue = pPipe->pRead->ItemVal;
					break;
				default:
					sRet = -3;
					break;
			}
			/* Lesezeiger versetzen */
			if( pPipe->pRead == pPipe->pLast ) {
				pPipe->pRead = pPipe->pFirst;
			}
			else {
				pPipe->pRead++;
			}
		} /* Meldung in Pipe */
		else {	/* Keine Meldung in Pipe */
			sRet = 0;	/* Pipe ist leer */
		}
	}
	return( sRet );
}

/*-----------------------------------------------------------------------------
// CliAktValToCabVal
// Setzt Cab.LastVal auf AktVal aus Alias-PV
// = Hilfsfunktion fuer CliItemLink() und CliItemLinkAll()
//
// LastEdit:
//		24.07.03/RES	Erstversion erstellt
//
// inputs:	pDtProps	Zeiger auf DT-Props des aktuellen Datentyps
//			pDtDesc		Zeiger auf DT-Desc des aktuellen Datentyps
//			pPab		Zeiger auf Datenpunkt in PAB
//			pCab		Zeiger auf Item in CAB
//			ItemIdx		Item-Index
// outputs:
// return:	  0 Aktuellen Wert aus Alias-PV erfolgreich auf Cab.LastVal kopiert
//			 -1 Keine Alias-PV, d.h. Leiche im PAB
//---------------------------------------------------------------------------*/
short CliAktValToCabVal( DtProps_Typ *pDtProps, DtDesc_Typ *pDtDesc, unsigned char *pPab, CabItemEntry_Typ *pCab, unsigned char ItemIdx )
{
	unsigned char	*pAlias;
	unsigned char	*pAktVal;

	/* Aktuellen Wert aus Alias-PV als LastVal ins CAB schreiben */
	pAlias = *(unsigned char **)( pPab + pDtProps->AliasPtrOff );
	if( pAlias == NULL ) {
		return( -1 );		/* Keine Alias-PV, d.h. Leiche im PAB */
	}
	pAktVal = pAlias + pDtDesc[ItemIdx].ItemOff;
	switch( abs( pDtDesc[ItemIdx].ItemLen ) ) {
		case 1:
			pCab->LastVal = ( unsigned long )*pAktVal;
			break;
		case 2:
			pCab->LastVal = ( unsigned long )*( unsigned short * )pAktVal;
			break;
		case 4:
			pCab->LastVal = *( unsigned long * )pAktVal;
			break;
	}
	return( 0 );
}
```

#### bksysgetpipe.c
```c
#ifdef _DEFAULT_INCLUDES
	#include <AsDefault.h>
#endif
/* bksysgetpipe.c ------------------------------------------------------------- */

#include <bur/plc.h>      /*some usefull macros for B&R pcc programming*/

#include <stdlib.h>

#include "bksys.h"

/*-----------------------------------------------------------------------------
// EvGetPipePtr
// Zeiger auf Event-Pipe ermitteln
// Last Edit:
//		13.07.99/RES
//		30.04.99/RES
//
// inputs:	UserID	Identity des zugehoerigen Dienstes
//          DtIdx	Datentyp-Index
//
// outputs: ppPipe	Zeiger auf Event-Pipe
//
// return:  Status: 0=kein Fehler, d.h. Pipe-Zeiger gueltig
//			       -1=unzulaessiger DtIdx
//				   -2=kein passender Event-Pipeblock gefunden
//				   -3=kein gueltiger Globals-Ptr
//---------------------------------------------------------------------------*/
short EvGetPipePtr( unsigned char UserID, unsigned char DtIdx, PipeHead_Typ** ppPipe )
{
	static Globals_Typ *pGlobals = NULL;

	short sRet = 0;
	EvPbHead_Typ* pEvBlock;

	/* Zeiger auf Struktur mit Zeigern auf Globaldaten initialisieren */
	if( pGlobals == NULL ) {
		GetGlobalsPtr( &pGlobals );
	}

	if( pGlobals != NULL ) {	/* Gueltiger Zeiger in pGlobals ? */
		if( DtIdx < DT_ANZ ) {	/* DtIdx zulaessig ? */
			/* Zugehoerigen Event-PipeBlock ermitteln */
			for( pEvBlock = pGlobals->pEvPipes; pEvBlock != NULL; pEvBlock = pEvBlock->pNext ) {
				if( pEvBlock->UserID == UserID ) {
					*ppPipe = pEvBlock->pDtPipe[DtIdx];
					break;	/* Event-Block gefunden ! */
				}
			}
			if( pEvBlock == NULL ) {
				sRet = NOEVBLKERR_NUM;	/* Kein EvPipeBlock mit angegebener UserID gefunden */
				ErrStatistics("", WARN, EC_SYS_BASE + NOEVBLKERR_NUM, 3, EC_SYS_BASE, NOEVBLKERR_TEXT );
			}
		}
		else {
			sRet = DTERR_NUM;	/* unzulaessiger DtIdx */
			ErrStatistics("", WARN, EC_SYS_BASE + DTERR_NUM, 3, EC_SYS_BASE, DTERR_TEXT );
		}
	}
	else {
		sRet = -3;
	}
	return( sRet );
}

/*-----------------------------------------------------------------------------
// CliGetPipePtr
// Zeiger auf Event-Pipe ermitteln
// Last Edit:
//		19.05.03/RES: Erstversion aus EvGetPipePtr() erzeugt
//
// inputs:	Client	Client
//          DtIdx	Datentyp-Index
//
// outputs: ppPipe	Zeiger auf Event-Pipe
//
// return:    0 kein Fehler, d.h. Pipe-Zeiger gueltig
//			 -1 Unzulaessiger Client
//			 -2 Unzulaessiger DtIdx
//			-10 Kein gueltiger Globals-Ptr
//			-11 Kein gueltiger Zeiger auf Pipeblock-Header
//			-12 Kein gueltiger PipeHead-Ptr
//---------------------------------------------------------------------------*/
short CliGetPipePtr( unsigned char Client, unsigned char DtIdx, CliPipeHead_Typ** ppPipe )
{
	static Globals_Typ	*pGlobals = NULL;

	short 				sRet = 0;
	CliPbHead_Typ 		*pPbHead;			/* Zeiger auf Client-Pipeblock-Header */

	/* Zeiger auf Struktur mit Zeigern auf Globaldaten initialisieren */
	if( pGlobals == NULL ) {
		GetGlobalsPtr( &pGlobals );
	}

	if( pGlobals != NULL ) {	/* Gueltiger Zeiger in pGlobals ? */
		if( Client < pGlobals->pCab->ClientAnz ) {
			pPbHead = pGlobals->pCab->pClientPb[Client];	/* Zeiger auf PipeBlock des angegebenen Clients ermitteln */
			if( pPbHead != 0 ) {
				if( DtIdx < DT_ANZ ) {	/* DtIdx zulaessig ? */
					*ppPipe = pPbHead->pDtPipe[DtIdx];	/* Zeiger auf Pipe-Header ermitteln */
					if( *ppPipe != 0 ) {
						sRet = 0;	/* Gueltiger PipeHead-Ptr gefunden */
					}
					else {
						sRet = -12;	/* Kein gueltiger PipeHead-Ptr */
					}
				}
				else {
					sRet = -2;	/* Unzulaessiger DtIdx */
				}
			}
			else {
				sRet = -11;	/* Kein gueltiger Zeiger auf Pipeblock-Header */
			}
		}
		else {
			sRet = -1;	/* Unzulaessiger Client */
		}
	}
	else {
		sRet = -10;	/* Kein gueltiger Globals-Ptr */
	}
	return( sRet );
}
```

#### bksysall.c
```c
#ifdef _DEFAULT_INCLUDES
	#include <AsDefault.h>
#endif
/* bksysall.c ----------------------------------------------------------------- */

#include <bur/plc.h>      /*some usefull macros for B&R pcc programming*/
#include <sys_lib.h>

#include <stdlib.h>
#include <string.h>

#include "bksys.h"

/*-----------------------------------------------------------------------------
// ErrStatistics
// Fehlerbehandlungsroutine
// Last Edit:
//		28.06.00/RES:	Bei mehrzeiligen Eintraegen wird ab Zeile 2 die Zeilennummer eingetragen
//		12.05.00/RES:	ErrNum=0 wird nicht mehr statistisch erfasst
//						pErrPre eingefuehrt
//						Aufteilung langer ErrTexte auf mehrere Logbuch-Eintraege
//						wobei bedingte und unbedingte Umbrueche definiert werden koennen
//		23.12.99/RES
//		30.04.99/RES
//
// inputs:	ErrStat		Fehlerstatus: 0=Warn, 1=Err, 2=Err+Log, 3=Err+Log+HALT
//			ErrNum		Fehlernummer
//			ErrInfo		Fehlerinfo
//			pErrPre		Praefix zu Fehlertext (fuer jede Eintragszeile)
//			pErrText	Zeiger auf Fehlertext
//
// outputs:
//
// return:
//---------------------------------------------------------------------------*/
void ErrStatistics( unsigned char *pTaskName,
					unsigned char ErrStat, unsigned short ErrNum, unsigned long ErrInfo,
					unsigned char *pErrPre, unsigned char *pErrText )
{
	static Stats_Typ *pStats = NULL;
	static short ErrFlag = 0;
	unsigned short LogErrNo;
	long lPtr, lVarLen;
	char szText[ERRTEXT_MAXLEN + 1];				/* Puffer fuer Fehlertext */
	char *pRead, *pWrite, *pStart, *pReadTemp;		/* Diverse Textzeiger */
	char buffer[64];
	short sByteAnz, sRest, sTextLen, sLine, sReadyText, sReadyLine, sSearchCount, sSearchCountMax;
	short sCutFlag = 0;		/* Trenn-Flag fuer Anzeige des Trennzeichens am Zeilenanfang */

	LogErrNo = EC_BK2_BASE + ErrNum;	/* Fehlernummer fuer Logbuch und LastErr sowie LastWarn */

	if( pStats == NULL ) {	/* Zeiger noch nicht bekannt ? */
		/* Zeiger auf Statistikstruktur ermitteln */
		strcpy(buffer, pTaskName);
		strcat(buffer, ":SYS_Statistic");
		if( !PV_xgetadr( buffer, &lPtr, &lVarLen ) ) {
			pStats = (Stats_Typ *)lPtr;
		}
		else {	/* SYS_Statistic nicht bekannt */
			if( ErrFlag == 0 ) {
				ERRxwarning( EC_BK2_BASE + EC_SYS_BASE + NOVALIDSTATSPTR_NUM, 0, NOVALIDSTATSPTR_TEXT );
				ErrFlag = 1;
			}
		}
	}
	if( pStats != NULL ) {	/* Zeiger bekannt ? */
		switch(ErrStat) {
			case WARN:	/* Warnmeldung */
				if( ErrNum > 0 ) {
					pStats->LastWarn = LogErrNo;
				}
				break;
			case ERR:	/* Fehlermeldung ohne Logbucheintrag */
				if( ErrNum > 0 ) {
					pStats->LastErr = LogErrNo;
				}
				break;
			case ERRLOG:		/* Fehlermeldung mit Logbucheintrag */
			case ERRLOGHALT:	/* Fehlermeldung mit Logbucheintrag und RPS-Halt */
				/* Fehlernummer eintragen */
				if( ErrNum > 0 ) {
					pStats->LastErr = LogErrNo;
				}
				/* Praefix in Textpuffer eintragen */
				sByteAnz = strlen( pErrPre );
				if( sByteAnz > 0 ) {	/* Praefix vorhanden! */
					if( sByteAnz >= ERRTEXT_MAXLEN ) {	/* Praefix laenger als Puffer ? */
						sByteAnz = ERRTEXT_MAXLEN - 1;
					}
					strncpy( szText, pErrPre, sByteAnz );
					pStart = szText + sByteAnz;
				}
				else {	/* Kein Praefix angegeben! */
					pStart = szText;
				}
				sTextLen = ERRTEXT_MAXLEN - ( pStart - szText );

				/* Fehlertext zeilenweise in Textpuffer eintragen und ins Logbuch schreiben */
				for( pRead = pErrText, sLine = 0, sReadyText = 0; !sReadyText && sLine < ERRTEXT_MAXLINES; sLine++ ) {
					pWrite = pStart;
					sRest = sTextLen;
					/* Zeilennummer fuer Folgezeilen einfuegen */
					if( sLine > 0 ) {
						if( sRest > 2 ) {	/* Nur, wenn mehr als 2 Zeichen fuer Nutztext zur Verfuegung! */
							*pWrite++ = '1' + sLine;
							sRest--;
						}
					}
					/* Prefic-Trennzeichen einfuegen */
					if( sRest > 2 ) {	/* Nur, wenn mehr als 2 Zeichen fuer Nutztext zur Verfuegung! */
						*pWrite++ = ':';
						sRest--;
					}

					/* Text fuer eine Meldezeile zusammenstellen */
					for( sReadyLine = 0; !sReadyLine && sRest > 0; sRest-- ) {
						/* Trennzeichen an Zeilenanfang einfuegen, wenn letzte Zeile abgeschnitten wurden */
						if( sCutFlag ) {
							sCutFlag = 0;
							if( sRest > 2 ) {	/* Nur, wenn mehr als 2 Zeichen fuer Nutztext zur Verfuegung! */
								*pWrite++ = CUT_SIGN;
								sRest--;
							}
						}
						/* Naechstes Lesezeichen auswerten */
						switch( *pRead  ) {
							case 0:		/* Ende des Fehlertextes erreicht */
								sReadyText = 1;
								sReadyLine = 1;
								break;
							case '\n':	/* Unbedingter Umbruch */
								sReadyLine = 1;
								pRead++;
								break;
							default:	/* Zu druckendes Textzeichen */
								if( sRest == 1 ) {	/* Zeilenende erreicht */
									switch( *( pRead + 1 ) ) {	/* Nachfolgendes Zeichen pruefen */
										case 0:		/* Ende des Fehlertextes erreicht */
											*pWrite++ = *pRead++;
											break;
										case '\n':	/* Unbedingter Umbruch */
										case '\t':	/* Bedingter Umbruch */
										case ' ':	/* Bedingter Umbruch */
											*pWrite++ = *pRead++;
											pRead++;	/* Trennzeichen ueberspringen */
											break;
										default:	/* Kein Trenn bzw. Endezeichen */
											/* Maximale Zeichenanzahl fuer nachfolgende Trennzeichensuche ermitteln */
											sSearchCountMax = ( SEARCH_COUNT_MAX < sTextLen ) ? SEARCH_COUNT_MAX : sTextLen;
											if( (short)strlen( pRead ) < sSearchCountMax ) {
												sSearchCountMax = strlen( pRead );
											}
											/* Letztes bedingtes Trennzeichen suchen */
											for( pReadTemp = pRead - 1, sSearchCount = 1; sSearchCount < sSearchCountMax; pReadTemp--, sSearchCount++ ) {
												if( *pReadTemp == ' ' || *pReadTemp == '\t' ) {
													break;	/* Trennzeichen gefunden => Suche abbrechen */
												}
											}
											if( sSearchCount < sSearchCountMax ) {	/* Suche vorzeitig abgebrochen, d.h. Trennzeichen gefunden */
												pRead -= sSearchCount - 1;	/* Lesezeiger auf Zeichen nach Trennzeichen setzen */
												pWrite -= sSearchCount;	/* Schreibzeiger auf Trennzeichen zuruecksetzen */
											}
											else {	/* Kein Trennzeichen gefunden => Zeile abschneiden */
												*pWrite++ = CUT_SIGN;	/* Kennzeichen fuer "harte" Trennung einfuegen */
												sCutFlag = 1;	/* Trenn-Flag fuer naechste Zeile merken */
											}
											break;
									} /* switch( *pRead ) */
								} /* if( sRest == 1 ) */
								else {	/* Noch nicht am Zeilenende ! */
									*pWrite++ = *pRead++;
								}
								break;
						} /* switch( *pRead ) */
					} /* Zeichenschleife */
					*pWrite = 0;	/* Zeichenkette abschliessen */

					/* Gesamte Zeile ins Logbuch schreiben */
					ERRxwarning( LogErrNo, bin_to_bcd_8( ErrInfo ), szText );

					/* Sonderfall "Textende gleich nach Zeilenende" pruefen */
					if( !sReadyText && *pRead == 0 ) {
						sReadyText = 1;	/*Textende-Flag setzen, um abschließende Leerzeile zu unterdruecken */
					}
				} /* Zeilenschleife */

				/* RPS anhalten ? */
				if( ErrStat == ERRLOGHALT ) {
					ERR_fatal( LogErrNo, bin_to_bcd_8( ErrInfo ) );
				}
				break;
			default:
				break;
		}
		/* Fehlerzaehler erhoehen */
		if( ErrNum > 0 && ErrNum < ERRCNTANZ ){
			if( pStats->ErrCount[ErrNum] < 65535 ) {
				pStats->ErrCount[ErrNum]++;
			}
		}
	}
}

/*-----------------------------------------------------------------------------
// ErrStatisticsX
// Erweiterte Fehlerbehandlungsroutine
// Variante 1: ErrBit entspricht Bitmuster in Fehlermaske ( 2-Byte )
// Last Edit:
//		10.05.00/RES:	pErrPre eingefuehrt
//		23.12.99/RES
//		19.05.99/RES
//
// inputs:  pErrMk		Zeiger auf Fehlermaske
//			ErrBit		Fehlerbit in Fehlermaske
// 			pSyErr  	Zeiger auf Systemfehlerzaehler
//			ErrStat1	Fehlerstatus 1. Auftreten des Fehlers: 0=Warn, 1=Err, 2=Err+Log, 3=Err+Log+HALT
//			ErrStatN	Fehlerstatus n. Auftreten des Fehlers: 0=Warn, 1=Err, 2=Err+Log, 3=Err+Log+HALT
//			ErrNum		Fehlernummer
//			ErrInfo		Fehlerinfo
//			pErrPre		Praefix zu Fehlertext (fuer jede Eintragszeile)
//			pErrText	Zeiger auf Fehlertext
//
// outputs:
//
// return:
//---------------------------------------------------------------------------*/
void ErrStatisticsX(unsigned char *pTaskName,
					unsigned short *pErrMk, unsigned short ErrBit, unsigned short *pSyErr,
					unsigned char ErrStat1, unsigned char ErrStatN, unsigned short ErrNum,
					unsigned long ErrInfo, unsigned char *pErrPre, unsigned char *pErrText )
{
	if( !(*pErrMk & ErrBit) ) {	/* Fehlerbit noch nicht gesetzt */
		*pErrMk |= ErrBit;
		ErrStatistics( pTaskName, ErrStat1, ErrNum, ErrInfo, pErrPre, pErrText );
	}
	else {
		ErrStatistics( pTaskName, ErrStatN, ErrNum, ErrInfo, pErrPre, pErrText );
	}
	if (pSyErr != NULL)
		*pSyErr += 1;
}

/*-----------------------------------------------------------------------------
// GetGlobalsPtr
// Liefert Zeiger auf Globaldatenstruktur
// Last Edit:
//		30.06.00/RES: ErrStatistics()-Aufruf bei Fehlern entfernt
//		19.07.99/RES
//		09.06.99/RES
//
// inputs:	-
// outputs: ppGlobals	Zeiger auf Globaldatenstruktur
// return:	-
//---------------------------------------------------------------------------*/
void GetGlobalsPtr( Globals_Typ **ppGlobals )
{
	static Globals_Typ *pGlobals = NULL;
	long lPtr, lVarLen;

	if( pGlobals == NULL ) {	/* Zeiger noch nicht bekannt ? */
		/* Zeiger auf Globaldatenstruktur ermitteln */
		if( !PV_xgetadr( "SYS_pGlobals", &lPtr, &lVarLen ) ) {
			pGlobals = *(Globals_Typ **)lPtr;
		}
		else {	/* SYS_pGlobals nicht gefunden */
			pGlobals = NULL;
		}
	}

	/* Zeiger zurueckliefern */
	*ppGlobals = pGlobals;
}
/*-----------------------------------------------------------------------------
// bin_to_bcd_8
// Wandelt Unsigned-long-Wert in 8-stellige BCD-Zahl (unsigned long) um
// Last Edit:
//		20.12.99/MKrz
//
// inputs:  value		Wert im Binaer-Format
//
// return:				Wert im BCD-Format
//---------------------------------------------------------------------------*/
unsigned long bin_to_bcd_8( unsigned long value )
{
	unsigned short	i;
	unsigned long	bcd = 0;
	unsigned long	tbin = 1;
	unsigned long	tbcd = 1;

	for (i=0; i<8; i++) {
		bcd += value/tbin % 10 * tbcd;
		tbin *= 10;
		tbcd *= 16;
	}
	return bcd;
}
```

### Program Logical/IEC103-Treiber/iec103 (ANSIC, version 6.40.0) - IEC 60870-5-103 Treiber
